KUKA KRL program: EPS_2_26115_SA7011_A_20260219035552.src

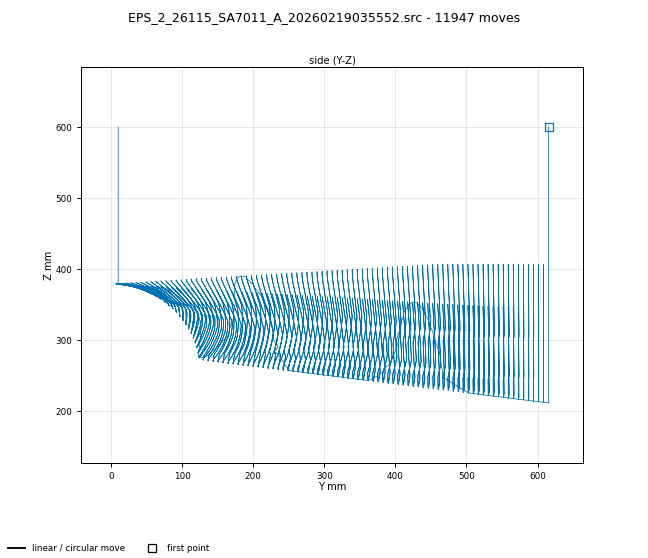
[picture p0: tool path of EPS_2_26115_SA7011_A_20260219035552.src, 11947 of 11949 moves have a stored position in this frame; points joined in program order, loops and branches not executed]
&ACCESS RVP
&REL 4
&COMMENT QRS 19112012
&PARAM EDITMASK = *
DEF PART()
EXT BAS (BAS_COMMAND :IN,REAL :IN )
INT I
BAS (#INITMOV,0 )

;KUKA QRS Post kuka4.cps  Date:22-06-2017 !

File_ID=3067

QRS_PRE_INIT()

;Init var - Until changes are made in qrs_pre_init
Outlet_Square_prg=0
Inlet_1_Square_prg=0
Inlet_2_Square_prg=0
Inlet_3_Square_prg=0
Inlet_4_Square_prg=0
Inlet_5_Square_prg=0

Outlet_1={X 0.000, Y 460.000, Z 306.500, B 0.000, E1 0.000 }
Inlet_1={X 0.000, Y 536.220, Z 246.500, B 0.000, E1 180.000 }
Outlet_1_type=201
Inlet_1_type=201
;QRS#1=Sidecore dimensions
;QRS#2=200-8" PVC SDR 35 Cut Back
;QRS#3=200-8" PVC SDR 35
;QRS#4=
;QRS#5=
;QRS#6=
;QRS#7=
;QRS#8=
;QRS#9=12-08 PSX
;QRS#10=12-08 PSX
;QRS#11=
;QRS#12=
;QRS#13=
;QRS#14=
;QRS#15=
;QRS#16=1220x127x686 2,25'
;QRS#17=EPS Height
;QRS#18=407
;QRS#19=*
;QRS#20= UPDATED VERSION 22-06-2017
;QRS#21=*
Outlet_Square=0100
Inlet_1_Square=0100
Inlet_2_Square=0
Inlet_3_Square=0
Inlet_4_Square=0
Inlet_5_Square=0
Mill_Square=1
Outlet_Square_Prg=214
Inlet_1_Square_prg=204

QRS_INIT()

$ADVANCE=5

; T1
PTP {E1 173.618,E2 173.618}
PTP {X 0,Y 615.492,A -85,B 0,C 180,E1 173.618,E2 173.618,E3 0,E4 0,E5 0,E6 0}
QRS_SPEED_INIT()
LIN {X 0,Y 615.492,Z 600,A -85,B 0,C 180,E1 173.618,E2 173.618,E3 0,E4 0,E5 0,E6 0} C_VEL
LIN {X 0,Y 615.492,Z 221.872,A -85,B 0,C 180,E1 173.618,E2 173.618} C_VEL
LIN {X 0,Y 615.492,Z 213.7,A -85,B 0,C 180,E1 173.618,E2 173.618} C_VEL
LIN {X 0,Y 615.48,Z 211.7,A -85,B 0,C 180,E1 173.432,E2 173.432} C_VEL
LIN {X 0,Y 615.497,Z 211.685,A -85,B 0,C 180,E1 170.801,E2 170.801} C_VEL
LIN {X 0,Y 615.486,Z 211.703,A -85,B 0,C 180,E1 168.139,E2 168.139} C_VEL
LIN {X 0,Y 615.448,Z 211.697,A -85,B 0,C 180,E1 165.45,E2 165.45} C_VEL
LIN {X 0,Y 615.468,Z 211.698,A -85,B 0,C 180,E1 162.729,E2 162.729} C_VEL
LIN {X 0,Y 615.465,Z 211.698,A -85,B 0,C 180,E1 159.966,E2 159.966} C_VEL
LIN {X 0,Y 615.489,Z 211.687,A -85,B 0,C 180,E1 157.155,E2 157.155} C_VEL
LIN {X 0,Y 615.481,Z 211.698,A -85,B 0,C 180,E1 154.284,E2 154.284} C_VEL
LIN {X 0,Y 615.466,Z 211.695,A -85,B 0,C 180,E1 151.554,E2 151.554} C_VEL
LIN {X 0,Y 615.449,Z 211.7,A -85,B 0,C 180,E1 148.921,E2 148.921} C_VEL
LIN {X 0,Y 615.453,Z 211.697,A -85,B 0,C 180,E1 146.471,E2 146.471} C_VEL
LIN {X 0,Y 615.489,Z 211.701,A -85,B 0,C 180,E1 144.167,E2 144.167} C_VEL
LIN {X 0,Y 615.48,Z 211.691,A -85,B 0,C 180,E1 141.931,E2 141.931} C_VEL
LIN {X 0,Y 615.493,Z 211.693,A -85,B 0,C 180,E1 139.394,E2 139.394} C_VEL
LIN {X 0,Y 615.44,Z 211.699,A -85,B 0,C 180,E1 136.751,E2 136.751} C_VEL
LIN {X 0,Y 615.483,Z 211.703,A -85,B 0,C 180,E1 133.997,E2 133.997} C_VEL
LIN {X 0,Y 615.468,Z 211.692,A -85,B 0,C 180,E1 131.476,E2 131.476} C_VEL
LIN {X 0,Y 615.489,Z 211.7,A -85,B 0,C 180,E1 128.905,E2 128.905} C_VEL
LIN {X 0,Y 615.472,Z 211.691,A -85,B 0,C 180,E1 126.426,E2 126.426} C_VEL
LIN {X 0,Y 615.493,Z 211.695,A -85,B 0,C 180,E1 125.616,E2 125.616} C_VEL
LIN {X 0,Y 615.455,Z 214.428,A -85,B 0,C 180,E1 123.239,E2 123.239} C_VEL
LIN {X 0,Y 615.428,Z 217.166,A -85,B 0,C 180,E1 120.923,E2 120.923} C_VEL
LIN {X 0,Y 615.496,Z 220.105,A -85,B 0,C 180,E1 118.451,E2 118.451} C_VEL
LIN {X 0,Y 615.445,Z 223.659,A -85,B 0,C 180,E1 115.718,E2 115.718} C_VEL
LIN {X 0,Y 615.442,Z 226.525,A -85,B 0,C 180,E1 113.558,E2 113.558} C_VEL
LIN {X 0,Y 615.45,Z 229.39,A -85,B 0,C 180,E1 111.434,E2 111.434} C_VEL
LIN {X 0,Y 615.496,Z 233.246,A -85,B 0,C 180,E1 108.606,E2 108.606} C_VEL
LIN {X 0,Y 615.457,Z 237.016,A -85,B 0,C 180,E1 105.906,E2 105.906} C_VEL
LIN {X 0,Y 615.495,Z 240.824,A -85,B 0,C 180,E1 103.201,E2 103.201} C_VEL
LIN {X 0,Y 615.481,Z 243.186,A -85,B 0,C 180,E1 101.548,E2 101.548} C_VEL
LIN {X 0,Y 615.491,Z 258.248,A -85,B 0,C 180,E1 101.193,E2 101.193} C_VEL
LIN {X 0,Y 615.496,Z 270.869,A -85,B 0,C 180,E1 100.753,E2 100.753} C_VEL
LIN {X 0,Y 615.468,Z 282.757,A -85,B 0,C 180,E1 100.195,E2 100.195} C_VEL
LIN {X 0,Y 615.497,Z 293.845,A -85,B 0,C 180,E1 99.53,E2 99.53} C_VEL
LIN {X 0,Y 615.498,Z 302.821,A -85,B 0,C 180,E1 98.868,E2 98.868} C_VEL
LIN {X 0,Y 615.498,Z 312.032,A -85,B 0,C 180,E1 98.041,E2 98.041} C_VEL
LIN {X 0,Y 615.499,Z 320.891,A -85,B 0,C 180,E1 97.058,E2 97.058} C_VEL
LIN {X 0,Y 615.497,Z 328.122,A -85,B 0,C 180,E1 96.063,E2 96.063} C_VEL
LIN {X 0,Y 615.497,Z 332.957,A -85,B 0,C 180,E1 95.241,E2 95.241} C_VEL
LIN {X 0,Y 615.493,Z 337.657,A -85,B 0,C 180,E1 94.257,E2 94.257} C_VEL
LIN {X 0,Y 615.495,Z 341.254,A -85,B 0,C 180,E1 93.273,E2 93.273} C_VEL
LIN {X 0,Y 615.496,Z 343.114,A -85,B 0,C 180,E1 92.618,E2 92.618} C_VEL
LIN {X 0,Y 615.497,Z 344.533,A -85,B 0,C 180,E1 91.963,E2 91.963} C_VEL
LIN {X 0,Y 615.496,Z 346.141,A -85,B 0,C 180,E1 90.654,E2 90.654} C_VEL
LIN {X 0,Y 615.494,Z 346.384,A -85,B 0,C 180,E1 90,E2 90} C_VEL
LIN {X 0,Y 615.495,Z 346.206,A -85,B 0,C 180,E1 89.346,E2 89.346} C_VEL
LIN {X 0,Y 615.496,Z 344.683,A -85,B 0,C 180,E1 88.037,E2 88.037} C_VEL
LIN {X 0,Y 615.498,Z 343.341,A -85,B 0,C 180,E1 87.382,E2 87.382} C_VEL
LIN {X 0,Y 615.496,Z 340.494,A -85,B 0,C 180,E1 86.399,E2 86.399} C_VEL
LIN {X 0,Y 615.498,Z 336.634,A -85,B 0,C 180,E1 85.416,E2 85.416} C_VEL
LIN {X 0,Y 615.498,Z 331.652,A -85,B 0,C 180,E1 84.43,E2 84.43} C_VEL
LIN {X 0,Y 615.497,Z 325.205,A -85,B 0,C 180,E1 83.417,E2 83.417} C_VEL
LIN {X 0,Y 615.497,Z 317.537,A -85,B 0,C 180,E1 82.455,E2 82.455} C_VEL
LIN {X 0,Y 615.498,Z 307.759,A -85,B 0,C 180,E1 81.464,E2 81.464} C_VEL
LIN {X 0,Y 615.498,Z 297.493,A -85,B 0,C 180,E1 80.636,E2 80.636} C_VEL
LIN {X 0,Y 615.469,Z 285.934,A -85,B 0,C 180,E1 79.888,E2 79.888} C_VEL
LIN {X 0,Y 615.492,Z 274.071,A -85,B 0,C 180,E1 79.293,E2 79.293} C_VEL
LIN {X 0,Y 615.486,Z 261.16,A -85,B 0,C 180,E1 78.807,E2 78.807} C_VEL
LIN {X 0,Y 615.486,Z 248.56,A -85,B 0,C 180,E1 78.473,E2 78.473} C_VEL
LIN {X 0,Y 615.483,Z 243.195,A -85,B 0,C 180,E1 78.369,E2 78.369} C_VEL
LIN {X 0,Y 615.466,Z 239.938,A -85,B 0,C 180,E1 76.077,E2 76.077} C_VEL
LIN {X 0,Y 615.49,Z 236.178,A -85,B 0,C 180,E1 73.413,E2 73.413} C_VEL
LIN {X 0,Y 615.472,Z 232.379,A -85,B 0,C 180,E1 70.662,E2 70.662} C_VEL
LIN {X 0,Y 615.458,Z 229.513,A -85,B 0,C 180,E1 68.567,E2 68.567} C_VEL
LIN {X 0,Y 615.465,Z 226.043,A -85,B 0,C 180,E1 65.997,E2 65.997} C_VEL
LIN {X 0,Y 615.494,Z 222.817,A -85,B 0,C 180,E1 63.556,E2 63.556} C_VEL
LIN {X 0,Y 615.475,Z 219.962,A -85,B 0,C 180,E1 61.341,E2 61.341} C_VEL
LIN {X 0,Y 615.429,Z 217.088,A -85,B 0,C 180,E1 58.924,E2 58.924} C_VEL
LIN {X 0,Y 615.471,Z 214.188,A -85,B 0,C 180,E1 56.469,E2 56.469} C_VEL
LIN {X 0,Y 615.496,Z 211.713,A -85,B 0,C 180,E1 54.385,E2 54.385} C_VEL
LIN {X 0,Y 615.485,Z 211.688,A -85,B 0,C 180,E1 51.931,E2 51.931} C_VEL
LIN {X 0,Y 615.487,Z 211.702,A -85,B 0,C 180,E1 49.393,E2 49.393} C_VEL
LIN {X 0,Y 615.455,Z 211.695,A -85,B 0,C 180,E1 46.752,E2 46.752} C_VEL
LIN {X 0,Y 615.466,Z 211.7,A -85,B 0,C 180,E1 43.995,E2 43.995} C_VEL
LIN {X 0,Y 615.447,Z 211.697,A -85,B 0,C 180,E1 41.477,E2 41.477} C_VEL
LIN {X 0,Y 615.49,Z 211.695,A -85,B 0,C 180,E1 38.904,E2 38.904} C_VEL
LIN {X 0,Y 615.486,Z 211.688,A -85,B 0,C 180,E1 36.425,E2 36.425} C_VEL
LIN {X 0,Y 615.492,Z 211.701,A -85,B 0,C 180,E1 34.022,E2 34.022} C_VEL
LIN {X 0,Y 615.442,Z 211.699,A -85,B 0,C 180,E1 31.688,E2 31.688} C_VEL
LIN {X 0,Y 615.439,Z 211.701,A -85,B 0,C 180,E1 29.409,E2 29.409} C_VEL
LIN {X 0,Y 615.471,Z 211.692,A -85,B 0,C 180,E1 26.445,E2 26.445} C_VEL
LIN {X 0,Y 615.478,Z 211.697,A -85,B 0,C 180,E1 24.006,E2 24.006} C_VEL
LIN {X 0,Y 615.471,Z 211.693,A -85,B 0,C 180,E1 21.433,E2 21.433} C_VEL
LIN {X 0,Y 615.491,Z 211.702,A -85,B 0,C 180,E1 18.605,E2 18.605} C_VEL
LIN {X 0,Y 615.434,Z 211.7,A -85,B 0,C 180,E1 15.907,E2 15.907} C_VEL
LIN {X 0,Y 615.495,Z 211.692,A -85,B 0,C 180,E1 13.201,E2 13.201} C_VEL
LIN {X 0,Y 615.472,Z 211.694,A -85,B 0,C 180,E1 10.527,E2 10.527} C_VEL
LIN {X 0,Y 615.473,Z 211.693,A -85,B 0,C 180,E1 7.876,E2 7.876} C_VEL
LIN {X 0,Y 615.497,Z 211.692,A -85,B 0,C 180,E1 5.241,E2 5.241} C_VEL
LIN {X 0,Y 615.437,Z 211.7,A -85,B 0,C 180,E1 2.618,E2 2.618} C_VEL
LIN {X 0,Y 615.477,Z 211.7,A -85,B 0,C 180,E1 0,E2 0} C_VEL
LIN {X 0,Y 615.483,Z 211.689,A -85,B 0,C 180,E1 -2.618,E2 -2.618} C_VEL
LIN {X 0,Y 615.496,Z 211.699,A -85,B 0,C 180,E1 -5.241,E2 -5.241} C_VEL
LIN {X 0,Y 615.466,Z 211.692,A -85,B 0,C 180,E1 -7.876,E2 -7.876} C_VEL
LIN {X 0,Y 615.485,Z 211.7,A -85,B 0,C 180,E1 -10.527,E2 -10.527} C_VEL
LIN {X 0,Y 615.437,Z 211.7,A -85,B 0,C 180,E1 -13.202,E2 -13.202} C_VEL
LIN {X 0,Y 615.495,Z 211.691,A -85,B 0,C 180,E1 -15.905,E2 -15.905} C_VEL
LIN {X 0,Y 615.481,Z 211.695,A -85,B 0,C 180,E1 -18.646,E2 -18.646} C_VEL
LIN {X 0,Y 615.468,Z 211.692,A -85,B 0,C 180,E1 -21.433,E2 -21.433} C_VEL
LIN {X 0,Y 615.475,Z 211.7,A -85,B 0,C 180,E1 -24.273,E2 -24.273} C_VEL
LIN {X 0,Y 615.436,Z 211.7,A -85,B 0,C 180,E1 -26.447,E2 -26.447} C_VEL
LIN {X 0,Y 615.452,Z 211.697,A -85,B 0,C 180,E1 -28.66,E2 -28.66} C_VEL
LIN {X 0,Y 615.488,Z 211.698,A -85,B 0,C 180,E1 -31.085,E2 -31.085} C_VEL
LIN {X 0,Y 615.495,Z 211.686,A -85,B 0,C 180,E1 -33.535,E2 -33.535} C_VEL
LIN {X 0,Y 615.464,Z 211.698,A -85,B 0,C 180,E1 -36.427,E2 -36.427} C_VEL
LIN {X 0,Y 615.458,Z 211.698,A -85,B 0,C 180,E1 -39.058,E2 -39.058} C_VEL
LIN {X 0,Y 615.484,Z 211.695,A -85,B 0,C 180,E1 -41.474,E2 -41.474} C_VEL
LIN {X 0,Y 615.463,Z 211.697,A -85,B 0,C 180,E1 -44.152,E2 -44.152} C_VEL
LIN {X 0,Y 615.484,Z 211.689,A -85,B 0,C 180,E1 -46.953,E2 -46.953} C_VEL
LIN {X 0,Y 615.479,Z 211.699,A -85,B 0,C 180,E1 -49.912,E2 -49.912} C_VEL
LIN {X 0,Y 615.446,Z 211.699,A -85,B 0,C 180,E1 -51.993,E2 -51.993} C_VEL
LIN {X 0,Y 615.46,Z 211.817,A -85,B 0,C 180,E1 -54.533,E2 -54.533} C_VEL
LIN {X 0,Y 615.471,Z 220.578,A -85,B 0,C 180,E1 -57.153,E2 -57.153} C_VEL
LIN {X 0,Y 615.452,Z 228.511,A -85,B 0,C 180,E1 -59.459,E2 -59.459} C_VEL
LIN {X 0,Y 615.48,Z 237.755,A -85,B 0,C 180,E1 -62.084,E2 -62.084} C_VEL
LIN {X 0,Y 615.488,Z 247.266,A -85,B 0,C 180,E1 -64.72,E2 -64.72} C_VEL
LIN {X 0,Y 615.475,Z 256.236,A -85,B 0,C 180,E1 -67.155,E2 -67.155} C_VEL
LIN {X 0,Y 615.49,Z 264.799,A -85,B 0,C 180,E1 -69.443,E2 -69.443} C_VEL
LIN {X 0,Y 615.49,Z 276.014,A -85,B 0,C 180,E1 -72.387,E2 -72.387} C_VEL
LIN {X 0,Y 615.479,Z 286.542,A -85,B 0,C 180,E1 -75.112,E2 -75.112} C_VEL
LIN {X 0,Y 615.444,Z 295.766,A -85,B 0,C 180,E1 -77.469,E2 -77.469} C_VEL
LIN {X 0,Y 615.498,Z 299.208,A -85,B 0,C 180,E1 -78.348,E2 -78.348} C_VEL
LIN {X 0,Y 615.497,Z 313.822,A -85,B 0,C 180,E1 -78.64,E2 -78.64} C_VEL
LIN {X 0,Y 615.451,Z 326.997,A -85,B 0,C 180,E1 -79.052,E2 -79.052} C_VEL
LIN {X 0,Y 615.438,Z 338.775,A -85,B 0,C 180,E1 -79.555,E2 -79.555} C_VEL
LIN {X 0,Y 615.482,Z 349.389,A -85,B 0,C 180,E1 -80.138,E2 -80.138} C_VEL
LIN {X 0,Y 615.498,Z 360.232,A -85,B 0,C 180,E1 -80.884,E2 -80.884} C_VEL
LIN {X 0,Y 615.497,Z 370.812,A -85,B 0,C 180,E1 -81.794,E2 -81.794} C_VEL
LIN {X 0,Y 615.498,Z 378.606,A -85,B 0,C 180,E1 -82.62,E2 -82.62} C_VEL
LIN {X 0,Y 615.496,Z 386.203,A -85,B 0,C 180,E1 -83.608,E2 -83.608} C_VEL
LIN {X 0,Y 615.498,Z 393.205,A -85,B 0,C 180,E1 -84.759,E2 -84.759} C_VEL
LIN {X 0,Y 615.494,Z 397.852,A -85,B 0,C 180,E1 -85.744,E2 -85.744} C_VEL
LIN {X 0,Y 615.494,Z 401.399,A -85,B 0,C 180,E1 -86.727,E2 -86.727} C_VEL
LIN {X 0,Y 615.497,Z 403.233,A -85,B 0,C 180,E1 -87.382,E2 -87.382} C_VEL
LIN {X 0,Y 615.5,Z 404.608,A -85,B 0,C 180,E1 -88.037,E2 -88.037} C_VEL
LIN {X 0,Y 615.496,Z 406.174,A -85,B 0,C 180,E1 -89.346,E2 -89.346} C_VEL
LIN {X 0,Y 615.494,Z 406.389,A -85,B 0,C 180,E1 -90,E2 -90} C_VEL
LIN {X 0,Y 615.495,Z 405.58,A -85,B 0,C 180,E1 -91.309,E2 -91.309} C_VEL
LIN {X 0,Y 615.5,Z 404.607,A -85,B 0,C 180,E1 -91.963,E2 -91.963} C_VEL
LIN {X 0,Y 615.497,Z 403.233,A -85,B 0,C 180,E1 -92.618,E2 -92.618} C_VEL
LIN {X 0,Y 615.496,Z 400.349,A -85,B 0,C 180,E1 -93.601,E2 -93.601} C_VEL
LIN {X 0,Y 615.498,Z 396.441,A -85,B 0,C 180,E1 -94.585,E2 -94.585} C_VEL
LIN {X 0,Y 615.499,Z 391.404,A -85,B 0,C 180,E1 -95.57,E2 -95.57} C_VEL
LIN {X 0,Y 615.497,Z 384.869,A -85,B 0,C 180,E1 -96.583,E2 -96.583} C_VEL
LIN {X 0,Y 615.497,Z 377.132,A -85,B 0,C 180,E1 -97.546,E2 -97.546} C_VEL
LIN {X 0,Y 615.498,Z 369.043,A -85,B 0,C 180,E1 -98.371,E2 -98.371} C_VEL
LIN {X 0,Y 615.499,Z 359.165,A -85,B 0,C 180,E1 -99.199,E2 -99.199} C_VEL
LIN {X 0,Y 615.471,Z 347.981,A -85,B 0,C 180,E1 -99.946,E2 -99.946} C_VEL
LIN {X 0,Y 615.437,Z 337.027,A -85,B 0,C 180,E1 -100.528,E2 -100.528} C_VEL
LIN {X 0,Y 615.457,Z 324.792,A -85,B 0,C 180,E1 -101.03,E2 -101.03} C_VEL
LIN {X 0,Y 615.499,Z 312.055,A -85,B 0,C 180,E1 -101.402,E2 -101.402} C_VEL
LIN {X 0,Y 615.498,Z 299.207,A -85,B 0,C 180,E1 -101.652,E2 -101.652} C_VEL
LIN {X 0,Y 615.454,Z 289.087,A -85,B 0,C 180,E1 -104.237,E2 -104.237} C_VEL
LIN {X 0,Y 615.491,Z 278.639,A -85,B 0,C 180,E1 -106.928,E2 -106.928} C_VEL
LIN {X 0,Y 615.482,Z 268.103,A -85,B 0,C 180,E1 -109.685,E2 -109.685} C_VEL
LIN {X 0,Y 615.49,Z 258.087,A -85,B 0,C 180,E1 -112.346,E2 -112.346} C_VEL
LIN {X 0,Y 615.477,Z 248.321,A -85,B 0,C 180,E1 -114.992,E2 -114.992} C_VEL
LIN {X 0,Y 615.492,Z 239.073,A -85,B 0,C 180,E1 -117.546,E2 -117.546} C_VEL
LIN {X 0,Y 615.456,Z 229.832,A -85,B 0,C 180,E1 -120.162,E2 -120.162} C_VEL
LIN {X 0,Y 615.445,Z 221.901,A -85,B 0,C 180,E1 -122.46,E2 -122.46} C_VEL
LIN {X 0,Y 615.492,Z 212.642,A -85,B 0,C 180,E1 -125.215,E2 -125.215} C_VEL
LIN {X 0,Y 615.455,Z 211.7,A -85,B 0,C 180,E1 -125.518,E2 -125.518} C_VEL
LIN {X 0,Y 615.448,Z 211.699,A -85,B 0,C 180,E1 -128.072,E2 -128.072} C_VEL
LIN {X 0,Y 615.491,Z 211.693,A -85,B 0,C 180,E1 -130.607,E2 -130.607} C_VEL
LIN {X 0,Y 615.48,Z 211.692,A -85,B 0,C 180,E1 -133.246,E2 -133.246} C_VEL
LIN {X 0,Y 615.459,Z 211.695,A -85,B 0,C 180,E1 -136.006,E2 -136.006} C_VEL
LIN {X 0,Y 615.48,Z 211.695,A -85,B 0,C 180,E1 -138.525,E2 -138.525} C_VEL
LIN {X 0,Y 615.446,Z 211.699,A -85,B 0,C 180,E1 -141.092,E2 -141.092} C_VEL
LIN {X 0,Y 615.462,Z 211.698,A -85,B 0,C 180,E1 -143.573,E2 -143.573} C_VEL
LIN {X 0,Y 615.495,Z 211.686,A -85,B 0,C 180,E1 -146.466,E2 -146.466} C_VEL
LIN {X 0,Y 615.491,Z 211.702,A -85,B 0,C 180,E1 -149.08,E2 -149.08} C_VEL
LIN {X 0,Y 615.45,Z 211.696,A -85,B 0,C 180,E1 -151.557,E2 -151.557} C_VEL
LIN {X 0,Y 615.471,Z 211.7,A -85,B 0,C 180,E1 -154.436,E2 -154.436} C_VEL
LIN {X 0,Y 615.469,Z 211.694,A -85,B 0,C 180,E1 -156.443,E2 -156.443} C_VEL
LIN {X 0,Y 615.466,Z 211.692,A -85,B 0,C 180,E1 -158.567,E2 -158.567} C_VEL
LIN {X 0,Y 615.483,Z 211.695,A -85,B 0,C 180,E1 -161.354,E2 -161.354} C_VEL
LIN {X 0,Y 615.495,Z 211.69,A -85,B 0,C 180,E1 -164.095,E2 -164.095} C_VEL
LIN {X 0,Y 615.442,Z 211.699,A -85,B 0,C 180,E1 -166.798,E2 -166.798} C_VEL
LIN {X 0,Y 615.48,Z 211.7,A -85,B 0,C 180,E1 -169.473,E2 -169.473} C_VEL
LIN {X 0,Y 615.467,Z 211.692,A -85,B 0,C 180,E1 -172.124,E2 -172.124} C_VEL
LIN {X 0,Y 615.495,Z 211.701,A -85,B 0,C 180,E1 -174.759,E2 -174.759} C_VEL
LIN {X 0,Y 615.484,Z 211.688,A -85,B 0,C 180,E1 -177.382,E2 -177.382} C_VEL
LIN {X 0,Y 615.479,Z 211.701,A -85,B 0,C 180,E1 -180,E2 -180} C_VEL
LIN {X 0,Y 615.435,Z 211.7,A -85,B 0,C 180,E1 -182.618,E2 -182.618} C_VEL
LIN {X 0,Y 615.497,Z 211.693,A -85,B 0,C 180,E1 -185.241,E2 -185.241} C_VEL
LIN {X 0,Y 615.48,Z 211.7,A -85,B 0,C 180,E1 -186.568,E2 -186.568} C_VEL
LIN {X 0,Y 614.812,Z 211.838,A -85,B 0,C 180,E1 -187.113,E2 -187.113} C_VEL
LIN {X 0,Y 611.989,Z 212.252,A -85,B 0,C 180,E1 -187.999,E2 -187.999} C_VEL
LIN {X 0,Y 609.599,Z 212.559,A -85,B 0,C 180,E1 -188.712,E2 -188.712} C_VEL
LIN {X 0,Y 608.558,Z 212.678,A -85,B 0,C 180,E1 -189.262,E2 -189.262} C_VEL
LIN {X 0,Y 608.466,Z 212.689,A -85,B 0,C 180,E1 -189.448,E2 -189.448} C_VEL
LIN {X 0,Y 608.458,Z 212.695,A -85,B 0,C 180,E1 -192,E2 -192} C_VEL
LIN {X 0,Y 608.422,Z 212.695,A -85,B 0,C 180,E1 -194.722,E2 -194.722} C_VEL
LIN {X 0,Y 608.428,Z 212.694,A -85,B 0,C 180,E1 -197.477,E2 -197.477} C_VEL
LIN {X 0,Y 608.433,Z 212.692,A -85,B 0,C 180,E1 -199.571,E2 -199.571} C_VEL
LIN {X 0,Y 608.483,Z 212.69,A -85,B 0,C 180,E1 -202.405,E2 -202.405} C_VEL
LIN {X 0,Y 608.457,Z 212.694,A -85,B 0,C 180,E1 -205.301,E2 -205.301} C_VEL
LIN {X 0,Y 608.437,Z 212.696,A -85,B 0,C 180,E1 -207.519,E2 -207.519} C_VEL
LIN {X 0,Y 608.406,Z 212.696,A -85,B 0,C 180,E1 -209.961,E2 -209.961} C_VEL
LIN {X 0,Y 608.47,Z 212.693,A -85,B 0,C 180,E1 -212.523,E2 -212.523} C_VEL
LIN {X 0,Y 608.439,Z 212.693,A -85,B 0,C 180,E1 -215.278,E2 -215.278} C_VEL
LIN {X 0,Y 608.465,Z 212.693,A -85,B 0,C 180,E1 -217.747,E2 -217.747} C_VEL
LIN {X 0,Y 608.449,Z 212.691,A -85,B 0,C 180,E1 -220.328,E2 -220.328} C_VEL
LIN {X 0,Y 608.424,Z 212.697,A -85,B 0,C 180,E1 -222.963,E2 -222.963} C_VEL
LIN {X 0,Y 608.441,Z 212.695,A -85,B 0,C 180,E1 -225.738,E2 -225.738} C_VEL
LIN {X 0,Y 608.442,Z 212.691,A -85,B 0,C 180,E1 -228.66,E2 -228.66} C_VEL
LIN {X 0,Y 608.471,Z 212.692,A -85,B 0,C 180,E1 -231.412,E2 -231.412} C_VEL
LIN {X 0,Y 608.451,Z 212.691,A -85,B 0,C 180,E1 -233.954,E2 -233.954} C_VEL
LIN {X 0,Y 608.437,Z 212.896,A -85,B 0,C 180,E1 -234.722,E2 -234.722} C_VEL
LIN {X 0,Y 608.403,Z 215.721,A -85,B 0,C 180,E1 -237.117,E2 -237.117} C_VEL
LIN {X 0,Y 608.435,Z 219.132,A -85,B 0,C 180,E1 -240.034,E2 -240.034} C_VEL
LIN {X 0,Y 608.39,Z 222.504,A -85,B 0,C 180,E1 -242.81,E2 -242.81} C_VEL
LIN {X 0,Y 608.413,Z 225.921,A -85,B 0,C 180,E1 -245.427,E2 -245.427} C_VEL
LIN {X 0,Y 608.385,Z 229.764,A -85,B 0,C 180,E1 -248.305,E2 -248.305} C_VEL
LIN {X 0,Y 608.388,Z 232.646,A -85,B 0,C 180,E1 -250.427,E2 -250.427} C_VEL
LIN {X 0,Y 608.417,Z 236.489,A -85,B 0,C 180,E1 -253.215,E2 -253.215} C_VEL
LIN {X 0,Y 608.394,Z 240.407,A -85,B 0,C 180,E1 -256.013,E2 -256.013} C_VEL
LIN {X 0,Y 608.423,Z 243.666,A -85,B 0,C 180,E1 -258.316,E2 -258.316} C_VEL
LIN {X 0,Y 608.535,Z 259.493,A -85,B 0,C 180,E1 -258.71,E2 -258.71} C_VEL
LIN {X 0,Y 608.518,Z 271.788,A -85,B 0,C 180,E1 -259.155,E2 -259.155} C_VEL
LIN {X 0,Y 608.467,Z 284.498,A -85,B 0,C 180,E1 -259.771,E2 -259.771} C_VEL
LIN {X 0,Y 608.487,Z 295.302,A -85,B 0,C 180,E1 -260.443,E2 -260.443} C_VEL
LIN {X 0,Y 608.477,Z 305.075,A -85,B 0,C 180,E1 -261.197,E2 -261.197} C_VEL
LIN {X 0,Y 608.46,Z 313.974,A -85,B 0,C 180,E1 -262.033,E2 -262.033} C_VEL
LIN {X 0,Y 608.465,Z 322.662,A -85,B 0,C 180,E1 -263.034,E2 -263.034} C_VEL
LIN {X 0,Y 608.439,Z 329.592,A -85,B 0,C 180,E1 -264.033,E2 -264.033} C_VEL
LIN {X 0,Y 608.436,Z 335.146,A -85,B 0,C 180,E1 -265.03,E2 -265.03} C_VEL
LIN {X 0,Y 608.434,Z 339.508,A -85,B 0,C 180,E1 -266.026,E2 -266.026} C_VEL
LIN {X 0,Y 608.425,Z 341.812,A -85,B 0,C 180,E1 -266.689,E2 -266.689} C_VEL
LIN {X 0,Y 608.425,Z 343.69,A -85,B 0,C 180,E1 -267.352,E2 -267.352} C_VEL
LIN {X 0,Y 608.442,Z 345.126,A -85,B 0,C 180,E1 -268.014,E2 -268.014} C_VEL
LIN {X 0,Y 608.439,Z 346.752,A -85,B 0,C 180,E1 -269.338,E2 -269.338} C_VEL
LIN {X 0,Y 608.434,Z 346.995,A -85,B 0,C 180,E1 -270,E2 -270} C_VEL
LIN {X 0,Y 608.438,Z 346.815,A -85,B 0,C 180,E1 -270.662,E2 -270.662} C_VEL
LIN {X 0,Y 608.441,Z 345.276,A -85,B 0,C 180,E1 -271.986,E2 -271.986} C_VEL
LIN {X 0,Y 608.427,Z 343.919,A -85,B 0,C 180,E1 -272.648,E2 -272.648} C_VEL
LIN {X 0,Y 608.449,Z 341.042,A -85,B 0,C 180,E1 -273.642,E2 -273.642} C_VEL
LIN {X 0,Y 608.433,Z 337.143,A -85,B 0,C 180,E1 -274.638,E2 -274.638} C_VEL
LIN {X 0,Y 608.449,Z 332.112,A -85,B 0,C 180,E1 -275.634,E2 -275.634} C_VEL
LIN {X 0,Y 608.442,Z 325.795,A -85,B 0,C 180,E1 -276.633,E2 -276.633} C_VEL
LIN {X 0,Y 608.475,Z 317.879,A -85,B 0,C 180,E1 -277.633,E2 -277.633} C_VEL
LIN {X 0,Y 608.472,Z 308.036,A -85,B 0,C 180,E1 -278.636,E2 -278.636} C_VEL
LIN {X 0,Y 608.481,Z 297.714,A -85,B 0,C 180,E1 -279.473,E2 -279.473} C_VEL
LIN {X 0,Y 608.466,Z 286.1,A -85,B 0,C 180,E1 -280.229,E2 -280.229} C_VEL
LIN {X 0,Y 608.509,Z 274.203,A -85,B 0,C 180,E1 -280.831,E2 -280.831} C_VEL
LIN {X 0,Y 608.529,Z 261.262,A -85,B 0,C 180,E1 -281.323,E2 -281.323} C_VEL
LIN {X 0,Y 608.535,Z 248.645,A -85,B 0,C 180,E1 -281.66,E2 -281.66} C_VEL
LIN {X 0,Y 608.427,Z 243.674,A -85,B 0,C 180,E1 -281.768,E2 -281.768} C_VEL
LIN {X 0,Y 608.418,Z 240.46,A -85,B 0,C 180,E1 -284.039,E2 -284.039} C_VEL
LIN {X 0,Y 608.418,Z 236.615,A -85,B 0,C 180,E1 -286.785,E2 -286.785} C_VEL
LIN {X 0,Y 608.395,Z 232.77,A -85,B 0,C 180,E1 -289.573,E2 -289.573} C_VEL
LIN {X 0,Y 608.389,Z 229.885,A -85,B 0,C 180,E1 -291.695,E2 -291.695} C_VEL
LIN {X 0,Y 608.416,Z 226.04,A -85,B 0,C 180,E1 -294.573,E2 -294.573} C_VEL
LIN {X 0,Y 608.398,Z 222.194,A -85,B 0,C 180,E1 -297.521,E2 -297.521} C_VEL
LIN {X 0,Y 608.437,Z 219.24,A -85,B 0,C 180,E1 -299.966,E2 -299.966} C_VEL
LIN {X 0,Y 608.397,Z 215.825,A -85,B 0,C 180,E1 -302.883,E2 -302.883} C_VEL
LIN {X 0,Y 608.436,Z 213.001,A -85,B 0,C 180,E1 -305.278,E2 -305.278} C_VEL
LIN {X 0,Y 608.478,Z 212.694,A -85,B 0,C 180,E1 -307.159,E2 -307.159} C_VEL
LIN {X 0,Y 608.449,Z 212.692,A -85,B 0,C 180,E1 -309.442,E2 -309.442} C_VEL
LIN {X 0,Y 608.469,Z 212.696,A -85,B 0,C 180,E1 -312.335,E2 -312.335} C_VEL
LIN {X 0,Y 608.414,Z 212.695,A -85,B 0,C 180,E1 -314.8,E2 -314.8} C_VEL
LIN {X 0,Y 608.468,Z 212.693,A -85,B 0,C 180,E1 -317.665,E2 -317.665} C_VEL
LIN {X 0,Y 608.447,Z 212.696,A -85,B 0,C 180,E1 -320.706,E2 -320.706} C_VEL
LIN {X 0,Y 608.451,Z 212.692,A -85,B 0,C 180,E1 -323.085,E2 -323.085} C_VEL
LIN {X 0,Y 608.472,Z 212.689,A -85,B 0,C 180,E1 -325.531,E2 -325.531} C_VEL
LIN {X 0,Y 608.459,Z 212.694,A -85,B 0,C 180,E1 -327.905,E2 -327.905} C_VEL
LIN {X 0,Y 608.419,Z 212.694,A -85,B 0,C 180,E1 -330.218,E2 -330.218} C_VEL
LIN {X 0,Y 608.461,Z 212.697,A -85,B 0,C 180,E1 -332.797,E2 -332.797} C_VEL
LIN {X 0,Y 608.45,Z 212.69,A -85,B 0,C 180,E1 -335.429,E2 -335.429} C_VEL
LIN {X 0,Y 608.463,Z 212.692,A -85,B 0,C 180,E1 -338.308,E2 -338.308} C_VEL
LIN {X 0,Y 608.476,Z 212.694,A -85,B 0,C 180,E1 -341.284,E2 -341.284} C_VEL
LIN {X 0,Y 608.416,Z 212.695,A -85,B 0,C 180,E1 -343.905,E2 -343.905} C_VEL
LIN {X 0,Y 608.464,Z 212.695,A -85,B 0,C 180,E1 -346.643,E2 -346.643} C_VEL
LIN {X 0,Y 608.453,Z 212.691,A -85,B 0,C 180,E1 -349.35,E2 -349.35} C_VEL
LIN {X 0,Y 608.469,Z 212.69,A -85,B 0,C 180,E1 -352.033,E2 -352.033} C_VEL
LIN {X 0,Y 608.473,Z 212.691,A -85,B 0,C 180,E1 -354.698,E2 -354.698} C_VEL
LIN {X 0,Y 608.435,Z 212.693,A -85,B 0,C 180,E1 -357.352,E2 -357.352} C_VEL
LIN {X 0,Y 608.469,Z 212.693,A -85,B 0,C 180,E1 -360,E2 -360} C_VEL
LIN {X 0,Y 608.475,Z 212.687,A -85,B 0,C 180,E1 -362.648,E2 -362.648} C_VEL
LIN {X 0,Y 608.473,Z 212.696,A -85,B 0,C 180,E1 -365.302,E2 -365.302} C_VEL
LIN {X 0,Y 608.437,Z 212.692,A -85,B 0,C 180,E1 -367.967,E2 -367.967} C_VEL
LIN {X 0,Y 608.45,Z 212.695,A -85,B 0,C 180,E1 -370.65,E2 -370.65} C_VEL
LIN {X 0,Y 608.432,Z 212.694,A -85,B 0,C 180,E1 -373.357,E2 -373.357} C_VEL
LIN {X 0,Y 608.461,Z 212.69,A -85,B 0,C 180,E1 -376.094,E2 -376.094} C_VEL
LIN {X 0,Y 608.454,Z 212.697,A -85,B 0,C 180,E1 -378.87,E2 -378.87} C_VEL
LIN {X 0,Y 608.461,Z 212.689,A -85,B 0,C 180,E1 -381.692,E2 -381.692} C_VEL
LIN {X 0,Y 608.429,Z 212.695,A -85,B 0,C 180,E1 -384.572,E2 -384.572} C_VEL
LIN {X 0,Y 608.455,Z 212.693,A -85,B 0,C 180,E1 -387.202,E2 -387.202} C_VEL
LIN {X 0,Y 608.445,Z 212.691,A -85,B 0,C 180,E1 -389.967,E2 -389.967} C_VEL
LIN {X 0,Y 608.462,Z 212.695,A -85,B 0,C 180,E1 -392.522,E2 -392.522} C_VEL
LIN {X 0,Y 608.442,Z 212.692,A -85,B 0,C 180,E1 -395.278,E2 -395.278} C_VEL
LIN {X 0,Y 608.456,Z 212.698,A -85,B 0,C 180,E1 -397.747,E2 -397.747} C_VEL
LIN {X 0,Y 608.404,Z 212.696,A -85,B 0,C 180,E1 -400.323,E2 -400.323} C_VEL
LIN {X 0,Y 608.457,Z 212.697,A -85,B 0,C 180,E1 -402.96,E2 -402.96} C_VEL
LIN {X 0,Y 608.445,Z 212.692,A -85,B 0,C 180,E1 -405.737,E2 -405.737} C_VEL
LIN {X 0,Y 608.452,Z 212.691,A -85,B 0,C 180,E1 -408.659,E2 -408.659} C_VEL
LIN {X 0,Y 608.435,Z 212.701,A -85,B 0,C 180,E1 -411.409,E2 -411.409} C_VEL
LIN {X 0,Y 608.429,Z 212.694,A -85,B 0,C 180,E1 -413.957,E2 -413.957} C_VEL
LIN {X 0,Y 608.446,Z 212.814,A -85,B 0,C 180,E1 -414.367,E2 -414.367} C_VEL
LIN {X 0,Y 608.529,Z 220.592,A -85,B 0,C 180,E1 -416.73,E2 -416.73} C_VEL
LIN {X 0,Y 608.481,Z 229.86,A -85,B 0,C 180,E1 -419.456,E2 -419.456} C_VEL
LIN {X 0,Y 608.494,Z 239.127,A -85,B 0,C 180,E1 -422.11,E2 -422.11} C_VEL
LIN {X 0,Y 608.479,Z 248.394,A -85,B 0,C 180,E1 -424.7,E2 -424.7} C_VEL
LIN {X 0,Y 608.48,Z 258.986,A -85,B 0,C 180,E1 -427.595,E2 -427.595} C_VEL
LIN {X 0,Y 608.457,Z 269.577,A -85,B 0,C 180,E1 -430.43,E2 -430.43} C_VEL
LIN {X 0,Y 608.45,Z 280.168,A -85,B 0,C 180,E1 -433.216,E2 -433.216} C_VEL
LIN {X 0,Y 608.437,Z 290.892,A -85,B 0,C 180,E1 -435.996,E2 -435.996} C_VEL
LIN {X 0,Y 608.437,Z 299.572,A -85,B 0,C 180,E1 -438.222,E2 -438.222} C_VEL
LIN {X 0,Y 608.55,Z 313.095,A -85,B 0,C 180,E1 -438.488,E2 -438.488} C_VEL
LIN {X 0,Y 608.486,Z 325.53,A -85,B 0,C 180,E1 -438.865,E2 -438.865} C_VEL
LIN {X 0,Y 608.444,Z 337.172,A -85,B 0,C 180,E1 -439.35,E2 -439.35} C_VEL
LIN {X 0,Y 608.471,Z 349.579,A -85,B 0,C 180,E1 -440.023,E2 -440.023} C_VEL
LIN {X 0,Y 608.483,Z 360.474,A -85,B 0,C 180,E1 -440.778,E2 -440.778} C_VEL
LIN {X 0,Y 608.475,Z 371.112,A -85,B 0,C 180,E1 -441.699,E2 -441.699} C_VEL
LIN {X 0,Y 608.471,Z 378.961,A -85,B 0,C 180,E1 -442.534,E2 -442.534} C_VEL
LIN {X 0,Y 608.461,Z 386.287,A -85,B 0,C 180,E1 -443.485,E2 -443.485} C_VEL
LIN {X 0,Y 608.451,Z 391.866,A -85,B 0,C 180,E1 -444.366,E2 -444.366} C_VEL
LIN {X 0,Y 608.432,Z 396.95,A -85,B 0,C 180,E1 -445.362,E2 -445.362} C_VEL
LIN {X 0,Y 608.449,Z 400.896,A -85,B 0,C 180,E1 -446.358,E2 -446.358} C_VEL
LIN {X 0,Y 608.425,Z 403.809,A -85,B 0,C 180,E1 -447.352,E2 -447.352} C_VEL
LIN {X 0,Y 608.444,Z 405.201,A -85,B 0,C 180,E1 -448.014,E2 -448.014} C_VEL
LIN {X 0,Y 608.438,Z 406.783,A -85,B 0,C 180,E1 -449.338,E2 -449.338} C_VEL
LIN {X 0,Y 608.434,Z 407,A -85,B 0,C 180,E1 -450,E2 -450} C_VEL
LIN {X 0,Y 608.448,Z 406.184,A -85,B 0,C 180,E1 -451.324,E2 -451.324} C_VEL
LIN {X 0,Y 608.444,Z 405.201,A -85,B 0,C 180,E1 -451.986,E2 -451.986} C_VEL
LIN {X 0,Y 608.425,Z 403.809,A -85,B 0,C 180,E1 -452.648,E2 -452.648} C_VEL
LIN {X 0,Y 608.449,Z 400.896,A -85,B 0,C 180,E1 -453.643,E2 -453.643} C_VEL
LIN {X 0,Y 608.432,Z 396.949,A -85,B 0,C 180,E1 -454.638,E2 -454.638} C_VEL
LIN {X 0,Y 608.438,Z 390.876,A -85,B 0,C 180,E1 -455.801,E2 -455.801} C_VEL
LIN {X 0,Y 608.462,Z 384.234,A -85,B 0,C 180,E1 -456.799,E2 -456.799} C_VEL
LIN {X 0,Y 608.456,Z 375.988,A -85,B 0,C 180,E1 -457.8,E2 -457.8} C_VEL
LIN {X 0,Y 608.472,Z 367.534,A -85,B 0,C 180,E1 -458.636,E2 -458.636} C_VEL
LIN {X 0,Y 608.48,Z 357.088,A -85,B 0,C 180,E1 -459.474,E2 -459.474} C_VEL
LIN {X 0,Y 608.482,Z 346.752,A -85,B 0,C 180,E1 -460.145,E2 -460.145} C_VEL
LIN {X 0,Y 608.463,Z 335.871,A -85,B 0,C 180,E1 -460.712,E2 -460.712} C_VEL
LIN {X 0,Y 608.492,Z 324.095,A -85,B 0,C 180,E1 -461.186,E2 -461.186} C_VEL
LIN {X 0,Y 608.551,Z 311.259,A -85,B 0,C 180,E1 -461.555,E2 -461.555} C_VEL
LIN {X 0,Y 608.439,Z 299.53,A -85,B 0,C 180,E1 -461.789,E2 -461.789} C_VEL
LIN {X 0,Y 608.405,Z 289.435,A -85,B 0,C 180,E1 -464.381,E2 -464.381} C_VEL
LIN {X 0,Y 608.45,Z 280.167,A -85,B 0,C 180,E1 -466.784,E2 -466.784} C_VEL
LIN {X 0,Y 608.457,Z 269.576,A -85,B 0,C 180,E1 -469.571,E2 -469.571} C_VEL
LIN {X 0,Y 608.464,Z 258.723,A -85,B 0,C 180,E1 -472.477,E2 -472.477} C_VEL
LIN {X 0,Y 608.479,Z 248.394,A -85,B 0,C 180,E1 -475.3,E2 -475.3} C_VEL
LIN {X 0,Y 608.496,Z 239.126,A -85,B 0,C 180,E1 -477.89,E2 -477.89} C_VEL
LIN {X 0,Y 608.481,Z 229.859,A -85,B 0,C 180,E1 -480.545,E2 -480.545} C_VEL
LIN {X 0,Y 608.528,Z 220.591,A -85,B 0,C 180,E1 -483.27,E2 -483.27} C_VEL
LIN {X 0,Y 608.438,Z 212.695,A -85,B 0,C 180,E1 -485.685,E2 -485.685} C_VEL
LIN {X 0,Y 608.443,Z 212.695,A -85,B 0,C 180,E1 -488.237,E2 -488.237} C_VEL
LIN {X 0,Y 608.448,Z 212.691,A -85,B 0,C 180,E1 -491.178,E2 -491.178} C_VEL
LIN {X 0,Y 608.466,Z 212.694,A -85,B 0,C 180,E1 -493.87,E2 -493.87} C_VEL
LIN {X 0,Y 608.483,Z 212.688,A -85,B 0,C 180,E1 -496.69,E2 -496.69} C_VEL
LIN {X 0,Y 608.45,Z 212.699,A -85,B 0,C 180,E1 -498.823,E2 -498.823} C_VEL
LIN {X 0,Y 608.417,Z 212.696,A -85,B 0,C 180,E1 -501.766,E2 -501.766} C_VEL
LIN {X 0,Y 608.45,Z 212.699,A -85,B 0,C 180,E1 -503.955,E2 -503.955} C_VEL
LIN {X 0,Y 608.47,Z 212.688,A -85,B 0,C 180,E1 -506.33,E2 -506.33} C_VEL
LIN {X 0,Y 608.451,Z 212.693,A -85,B 0,C 180,E1 -508.733,E2 -508.733} C_VEL
LIN {X 0,Y 608.445,Z 212.692,A -85,B 0,C 180,E1 -511.386,E2 -511.386} C_VEL
LIN {X 0,Y 608.47,Z 212.695,A -85,B 0,C 180,E1 -514.281,E2 -514.281} C_VEL
LIN {X 0,Y 608.429,Z 212.693,A -85,B 0,C 180,E1 -516.875,E2 -516.875} C_VEL
LIN {X 0,Y 608.469,Z 212.696,A -85,B 0,C 180,E1 -519.322,E2 -519.322} C_VEL
LIN {X 0,Y 608.452,Z 212.69,A -85,B 0,C 180,E1 -521.828,E2 -521.828} C_VEL
LIN {X 0,Y 608.463,Z 212.695,A -85,B 0,C 180,E1 -524.594,E2 -524.594} C_VEL
LIN {X 0,Y 608.435,Z 212.694,A -85,B 0,C 180,E1 -526.643,E2 -526.643} C_VEL
LIN {X 0,Y 608.446,Z 212.695,A -85,B 0,C 180,E1 -529.35,E2 -529.35} C_VEL
LIN {X 0,Y 608.438,Z 212.692,A -85,B 0,C 180,E1 -532.033,E2 -532.033} C_VEL
LIN {X 0,Y 608.472,Z 212.695,A -85,B 0,C 180,E1 -534.698,E2 -534.698} C_VEL
LIN {X 0,Y 608.476,Z 212.687,A -85,B 0,C 180,E1 -537.352,E2 -537.352} C_VEL
LIN {X 0,Y 608.471,Z 212.694,A -85,B 0,C 180,E1 -540,E2 -540} C_VEL
LIN {X 0,Y 608.433,Z 212.693,A -85,B 0,C 180,E1 -542.648,E2 -542.648} C_VEL
LIN {X 0,Y 608.472,Z 212.691,A -85,B 0,C 180,E1 -545.302,E2 -545.302} C_VEL
LIN {X 0,Y 608.44,Z 212.694,A -85,B 0,C 180,E1 -547.968,E2 -547.968} C_VEL
LIN {X 0,Y 608.466,Z 212.689,A -85,B 0,C 180,E1 -549.448,E2 -549.448} C_VEL
LIN {X 0,Y 607.778,Z 212.78,A -85,B 0,C 180,E1 -550,E2 -550} C_VEL
LIN {X 0,Y 604.922,Z 213.136,A -85,B 0,C 180,E1 -550.897,E2 -550.897} C_VEL
LIN {X 0,Y 602.52,Z 213.434,A -85,B 0,C 180,E1 -551.619,E2 -551.619} C_VEL
LIN {X 0,Y 601.488,Z 213.561,A -85,B 0,C 180,E1 -552.175,E2 -552.175} C_VEL
LIN {X 0,Y 601.403,Z 213.57,A -85,B 0,C 180,E1 -552.364,E2 -552.364} C_VEL
LIN {X 0,Y 601.394,Z 213.572,A -85,B 0,C 180,E1 -554.898,E2 -554.898} C_VEL
LIN {X 0,Y 601.373,Z 213.572,A -85,B 0,C 180,E1 -557.689,E2 -557.689} C_VEL
LIN {X 0,Y 601.434,Z 213.57,A -85,B 0,C 180,E1 -560.522,E2 -560.522} C_VEL
LIN {X 0,Y 601.4,Z 213.571,A -85,B 0,C 180,E1 -563.411,E2 -563.411} C_VEL
LIN {X 0,Y 601.409,Z 213.571,A -85,B 0,C 180,E1 -565.865,E2 -565.865} C_VEL
LIN {X 0,Y 601.424,Z 213.569,A -85,B 0,C 180,E1 -568.627,E2 -568.627} C_VEL
LIN {X 0,Y 601.393,Z 213.57,A -85,B 0,C 180,E1 -571.728,E2 -571.728} C_VEL
LIN {X 0,Y 601.424,Z 213.573,A -85,B 0,C 180,E1 -574.119,E2 -574.119} C_VEL
LIN {X 0,Y 601.402,Z 213.569,A -85,B 0,C 180,E1 -576.583,E2 -576.583} C_VEL
LIN {X 0,Y 601.409,Z 213.575,A -85,B 0,C 180,E1 -579.127,E2 -579.127} C_VEL
LIN {X 0,Y 601.414,Z 213.567,A -85,B 0,C 180,E1 -581.766,E2 -581.766} C_VEL
LIN {X 0,Y 601.402,Z 213.573,A -85,B 0,C 180,E1 -584.532,E2 -584.532} C_VEL
LIN {X 0,Y 601.388,Z 213.573,A -85,B 0,C 180,E1 -587.412,E2 -587.412} C_VEL
LIN {X 0,Y 601.406,Z 213.569,A -85,B 0,C 180,E1 -590.004,E2 -590.004} C_VEL
LIN {X 0,Y 601.44,Z 213.568,A -85,B 0,C 180,E1 -592.618,E2 -592.618} C_VEL
LIN {X 0,Y 601.375,Z 213.806,A -85,B 0,C 180,E1 -594.891,E2 -594.891} C_VEL
LIN {X 0,Y 601.349,Z 216.8,A -85,B 0,C 180,E1 -597.479,E2 -597.479} C_VEL
LIN {X 0,Y 601.349,Z 219.549,A -85,B 0,C 180,E1 -599.865,E2 -599.865} C_VEL
LIN {X 0,Y 601.314,Z 222.827,A -85,B 0,C 180,E1 -602.657,E2 -602.657} C_VEL
LIN {X 0,Y 601.327,Z 225.921,A -85,B 0,C 180,E1 -605.118,E2 -605.118} C_VEL
LIN {X 0,Y 601.32,Z 229.764,A -85,B 0,C 180,E1 -608.037,E2 -608.037} C_VEL
LIN {X 0,Y 601.297,Z 232.647,A -85,B 0,C 180,E1 -610.187,E2 -610.187} C_VEL
LIN {X 0,Y 601.295,Z 235.529,A -85,B 0,C 180,E1 -612.308,E2 -612.308} C_VEL
LIN {X 0,Y 601.31,Z 238.412,A -85,B 0,C 180,E1 -614.406,E2 -614.406} C_VEL
LIN {X 0,Y 601.321,Z 242.256,A -85,B 0,C 180,E1 -617.169,E2 -617.169} C_VEL
LIN {X 0,Y 601.328,Z 243.667,A -85,B 0,C 180,E1 -618.176,E2 -618.176} C_VEL
LIN {X 0,Y 601.598,Z 247.38,A -85,B 0,C 180,E1 -618.267,E2 -618.267} C_VEL
LIN {X 0,Y 601.565,Z 259.674,A -85,B 0,C 180,E1 -618.583,E2 -618.583} C_VEL
LIN {X 0,Y 601.547,Z 272.824,A -85,B 0,C 180,E1 -619.072,E2 -619.072} C_VEL
LIN {X 0,Y 601.477,Z 284.51,A -85,B 0,C 180,E1 -619.65,E2 -619.65} C_VEL
LIN {X 0,Y 601.458,Z 295.308,A -85,B 0,C 180,E1 -620.33,E2 -620.33} C_VEL
LIN {X 0,Y 601.435,Z 305.082,A -85,B 0,C 180,E1 -621.093,E2 -621.093} C_VEL
LIN {X 0,Y 601.407,Z 313.979,A -85,B 0,C 180,E1 -621.939,E2 -621.939} C_VEL
LIN {X 0,Y 601.407,Z 322.666,A -85,B 0,C 180,E1 -622.952,E2 -622.952} C_VEL
LIN {X 0,Y 601.361,Z 329.596,A -85,B 0,C 180,E1 -623.962,E2 -623.962} C_VEL
LIN {X 0,Y 601.345,Z 335.148,A -85,B 0,C 180,E1 -624.971,E2 -624.971} C_VEL
LIN {X 0,Y 601.346,Z 339.51,A -85,B 0,C 180,E1 -625.979,E2 -625.979} C_VEL
LIN {X 0,Y 601.344,Z 341.814,A -85,B 0,C 180,E1 -626.65,E2 -626.65} C_VEL
LIN {X 0,Y 601.324,Z 343.692,A -85,B 0,C 180,E1 -627.32,E2 -627.32} C_VEL
LIN {X 0,Y 601.341,Z 345.127,A -85,B 0,C 180,E1 -627.991,E2 -627.991} C_VEL
LIN {X 0,Y 601.339,Z 346.752,A -85,B 0,C 180,E1 -629.33,E2 -629.33} C_VEL
LIN {X 0,Y 601.335,Z 346.996,A -85,B 0,C 180,E1 -630,E2 -630} C_VEL
LIN {X 0,Y 601.339,Z 346.815,A -85,B 0,C 180,E1 -630.67,E2 -630.67} C_VEL
LIN {X 0,Y 601.34,Z 345.276,A -85,B 0,C 180,E1 -632.009,E2 -632.009} C_VEL
LIN {X 0,Y 601.326,Z 343.917,A -85,B 0,C 180,E1 -632.679,E2 -632.679} C_VEL
LIN {X 0,Y 601.368,Z 341.04,A -85,B 0,C 180,E1 -633.685,E2 -633.685} C_VEL
LIN {X 0,Y 601.337,Z 337.141,A -85,B 0,C 180,E1 -634.693,E2 -634.693} C_VEL
LIN {X 0,Y 601.373,Z 332.11,A -85,B 0,C 180,E1 -635.701,E2 -635.701} C_VEL
LIN {X 0,Y 601.382,Z 325.792,A -85,B 0,C 180,E1 -636.711,E2 -636.711} C_VEL
LIN {X 0,Y 601.396,Z 317.874,A -85,B 0,C 180,E1 -637.723,E2 -637.723} C_VEL
LIN {X 0,Y 601.437,Z 308.03,A -85,B 0,C 180,E1 -638.738,E2 -638.738} C_VEL
LIN {X 0,Y 601.448,Z 297.709,A -85,B 0,C 180,E1 -639.585,E2 -639.585} C_VEL
LIN {X 0,Y 601.479,Z 286.089,A -85,B 0,C 180,E1 -640.349,E2 -640.349} C_VEL
LIN {X 0,Y 601.524,Z 274.192,A -85,B 0,C 180,E1 -640.959,E2 -640.959} C_VEL
LIN {X 0,Y 601.551,Z 261.247,A -85,B 0,C 180,E1 -641.456,E2 -641.456} C_VEL
LIN {X 0,Y 601.604,Z 248.622,A -85,B 0,C 180,E1 -641.797,E2 -641.797} C_VEL
LIN {X 0,Y 601.331,Z 243.673,A -85,B 0,C 180,E1 -641.909,E2 -641.909} C_VEL
LIN {X 0,Y 601.317,Z 240.459,A -85,B 0,C 180,E1 -644.208,E2 -644.208} C_VEL
LIN {X 0,Y 601.334,Z 236.614,A -85,B 0,C 180,E1 -646.989,E2 -646.989} C_VEL
LIN {X 0,Y 601.301,Z 232.769,A -85,B 0,C 180,E1 -649.813,E2 -649.813} C_VEL
LIN {X 0,Y 601.322,Z 229.885,A -85,B 0,C 180,E1 -651.963,E2 -651.963} C_VEL
LIN {X 0,Y 601.331,Z 226.039,A -85,B 0,C 180,E1 -654.882,E2 -654.882} C_VEL
LIN {X 0,Y 601.32,Z 222.899,A -85,B 0,C 180,E1 -657.344,E2 -657.344} C_VEL
LIN {X 0,Y 601.352,Z 219.647,A -85,B 0,C 180,E1 -660.168,E2 -660.168} C_VEL
LIN {X 0,Y 601.335,Z 216.694,A -85,B 0,C 180,E1 -662.702,E2 -662.702} C_VEL
LIN {X 0,Y 601.371,Z 213.909,A -85,B 0,C 180,E1 -665.108,E2 -665.108} C_VEL
LIN {X 0,Y 601.399,Z 213.57,A -85,B 0,C 180,E1 -666.583,E2 -666.583} C_VEL
LIN {X 0,Y 601.418,Z 213.571,A -85,B 0,C 180,E1 -669.126,E2 -669.126} C_VEL
LIN {X 0,Y 601.425,Z 213.566,A -85,B 0,C 180,E1 -671.765,E2 -671.765} C_VEL
LIN {X 0,Y 601.4,Z 213.57,A -85,B 0,C 180,E1 -674.532,E2 -674.532} C_VEL
LIN {X 0,Y 601.41,Z 213.575,A -85,B 0,C 180,E1 -677.41,E2 -677.41} C_VEL
LIN {X 0,Y 601.403,Z 213.568,A -85,B 0,C 180,E1 -680.004,E2 -680.004} C_VEL
LIN {X 0,Y 601.438,Z 213.572,A -85,B 0,C 180,E1 -682.618,E2 -682.618} C_VEL
LIN {X 0,Y 601.407,Z 213.568,A -85,B 0,C 180,E1 -685.067,E2 -685.067} C_VEL
LIN {X 0,Y 601.436,Z 213.569,A -85,B 0,C 180,E1 -687.484,E2 -687.484} C_VEL
LIN {X 0,Y 601.373,Z 213.574,A -85,B 0,C 180,E1 -689.861,E2 -689.861} C_VEL
LIN {X 0,Y 601.372,Z 213.572,A -85,B 0,C 180,E1 -692.13,E2 -692.13} C_VEL
LIN {X 0,Y 601.431,Z 213.57,A -85,B 0,C 180,E1 -694.382,E2 -694.382} C_VEL
LIN {X 0,Y 601.421,Z 213.569,A -85,B 0,C 180,E1 -696.59,E2 -696.59} C_VEL
LIN {X 0,Y 601.434,Z 213.57,A -85,B 0,C 180,E1 -699.478,E2 -699.478} C_VEL
LIN {X 0,Y 601.374,Z 213.572,A -85,B 0,C 180,E1 -702.311,E2 -702.311} C_VEL
LIN {X 0,Y 601.393,Z 213.573,A -85,B 0,C 180,E1 -705.102,E2 -705.102} C_VEL
LIN {X 0,Y 601.411,Z 213.57,A -85,B 0,C 180,E1 -707.857,E2 -707.857} C_VEL
LIN {X 0,Y 601.424,Z 213.566,A -85,B 0,C 180,E1 -710.584,E2 -710.584} C_VEL
LIN {X 0,Y 601.435,Z 213.572,A -85,B 0,C 180,E1 -713.345,E2 -713.345} C_VEL
LIN {X 0,Y 601.371,Z 213.572,A -85,B 0,C 180,E1 -715.979,E2 -715.979} C_VEL
LIN {X 0,Y 601.417,Z 213.572,A -85,B 0,C 180,E1 -718.661,E2 -718.661} C_VEL
LIN {X 0,Y 601.398,Z 213.57,A -85,B 0,C 180,E1 -721.339,E2 -721.339} C_VEL
LIN {X 0,Y 601.422,Z 213.57,A -85,B 0,C 180,E1 -723.35,E2 -723.35} C_VEL
LIN {X 0,Y 601.406,Z 213.568,A -85,B 0,C 180,E1 -726.037,E2 -726.037} C_VEL
LIN {X 0,Y 601.415,Z 213.575,A -85,B 0,C 180,E1 -728.738,E2 -728.738} C_VEL
LIN {X 0,Y 601.396,Z 213.569,A -85,B 0,C 180,E1 -731.459,E2 -731.459} C_VEL
LIN {X 0,Y 601.417,Z 213.569,A -85,B 0,C 180,E1 -734.206,E2 -734.206} C_VEL
LIN {X 0,Y 601.415,Z 213.571,A -85,B 0,C 180,E1 -736.986,E2 -736.986} C_VEL
LIN {X 0,Y 601.406,Z 213.568,A -85,B 0,C 180,E1 -739.809,E2 -739.809} C_VEL
LIN {X 0,Y 601.413,Z 213.571,A -85,B 0,C 180,E1 -742.683,E2 -742.683} C_VEL
LIN {X 0,Y 601.378,Z 213.571,A -85,B 0,C 180,E1 -744.88,E2 -744.88} C_VEL
LIN {X 0,Y 601.398,Z 213.574,A -85,B 0,C 180,E1 -747.359,E2 -747.359} C_VEL
LIN {X 0,Y 601.405,Z 213.568,A -85,B 0,C 180,E1 -750.165,E2 -750.165} C_VEL
LIN {X 0,Y 601.423,Z 213.573,A -85,B 0,C 180,E1 -752.715,E2 -752.715} C_VEL
LIN {X 0,Y 601.392,Z 213.57,A -85,B 0,C 180,E1 -755.111,E2 -755.111} C_VEL
LIN {X 0,Y 601.432,Z 213.568,A -85,B 0,C 180,E1 -757.419,E2 -757.419} C_VEL
LIN {X 0,Y 601.376,Z 213.573,A -85,B 0,C 180,E1 -759.998,E2 -759.998} C_VEL
LIN {X 0,Y 601.387,Z 213.575,A -85,B 0,C 180,E1 -762.673,E2 -762.673} C_VEL
LIN {X 0,Y 601.401,Z 213.569,A -85,B 0,C 180,E1 -765.479,E2 -765.479} C_VEL
LIN {X 0,Y 601.422,Z 213.569,A -85,B 0,C 180,E1 -768.407,E2 -768.407} C_VEL
LIN {X 0,Y 601.402,Z 213.57,A -85,B 0,C 180,E1 -770.872,E2 -770.872} C_VEL
LIN {X 0,Y 601.396,Z 213.576,A -85,B 0,C 180,E1 -773.416,E2 -773.416} C_VEL
LIN {X 0,Y 601.403,Z 213.688,A -85,B 0,C 180,E1 -774.158,E2 -774.158} C_VEL
LIN {X 0,Y 601.544,Z 219.268,A -85,B 0,C 180,E1 -775.889,E2 -775.889} C_VEL
LIN {X 0,Y 601.566,Z 228.022,A -85,B 0,C 180,E1 -778.523,E2 -778.523} C_VEL
LIN {X 0,Y 601.479,Z 237.803,A -85,B 0,C 180,E1 -781.375,E2 -781.375} C_VEL
LIN {X 0,Y 601.478,Z 247.454,A -85,B 0,C 180,E1 -784.12,E2 -784.12} C_VEL
LIN {X 0,Y 601.466,Z 256.338,A -85,B 0,C 180,E1 -786.592,E2 -786.592} C_VEL
LIN {X 0,Y 601.431,Z 266.929,A -85,B 0,C 180,E1 -789.478,E2 -789.478} C_VEL
LIN {X 0,Y 601.4,Z 277.52,A -85,B 0,C 180,E1 -792.312,E2 -792.312} C_VEL
LIN {X 0,Y 601.366,Z 288.112,A -85,B 0,C 180,E1 -795.101,E2 -795.101} C_VEL
LIN {X 0,Y 601.342,Z 298.703,A -85,B 0,C 180,E1 -797.856,E2 -797.856} C_VEL
LIN {X 0,Y 601.372,Z 299.53,A -85,B 0,C 180,E1 -798.071,E2 -798.071} C_VEL
LIN {X 0,Y 601.618,Z 311.268,A -85,B 0,C 180,E1 -798.311,E2 -798.311} C_VEL
LIN {X 0,Y 601.533,Z 324.353,A -85,B 0,C 180,E1 -798.692,E2 -798.692} C_VEL
LIN {X 0,Y 601.48,Z 335.262,A -85,B 0,C 180,E1 -799.133,E2 -799.133} C_VEL
LIN {X 0,Y 601.473,Z 346.756,A -85,B 0,C 180,E1 -799.736,E2 -799.736} C_VEL
LIN {X 0,Y 601.462,Z 358.253,A -85,B 0,C 180,E1 -800.5,E2 -800.5} C_VEL
LIN {X 0,Y 601.436,Z 367.537,A -85,B 0,C 180,E1 -801.262,E2 -801.262} C_VEL
LIN {X 0,Y 601.4,Z 375.99,A -85,B 0,C 180,E1 -802.108,E2 -802.108} C_VEL
LIN {X 0,Y 601.382,Z 384.236,A -85,B 0,C 180,E1 -803.12,E2 -803.12} C_VEL
LIN {X 0,Y 601.373,Z 390.877,A -85,B 0,C 180,E1 -804.131,E2 -804.131} C_VEL
LIN {X 0,Y 601.336,Z 396.95,A -85,B 0,C 180,E1 -805.307,E2 -805.307} C_VEL
LIN {X 0,Y 601.368,Z 400.896,A -85,B 0,C 180,E1 -806.315,E2 -806.315} C_VEL
LIN {X 0,Y 601.325,Z 403.809,A -85,B 0,C 180,E1 -807.321,E2 -807.321} C_VEL
LIN {X 0,Y 601.343,Z 405.202,A -85,B 0,C 180,E1 -807.991,E2 -807.991} C_VEL
LIN {X 0,Y 601.339,Z 406.784,A -85,B 0,C 180,E1 -809.33,E2 -809.33} C_VEL
LIN {X 0,Y 601.335,Z 407,A -85,B 0,C 180,E1 -810,E2 -810} C_VEL
LIN {X 0,Y 601.347,Z 406.184,A -85,B 0,C 180,E1 -811.339,E2 -811.339} C_VEL
LIN {X 0,Y 601.343,Z 405.201,A -85,B 0,C 180,E1 -812.009,E2 -812.009} C_VEL
LIN {X 0,Y 601.325,Z 403.809,A -85,B 0,C 180,E1 -812.68,E2 -812.68} C_VEL
LIN {X 0,Y 601.368,Z 400.896,A -85,B 0,C 180,E1 -813.685,E2 -813.685} C_VEL
LIN {X 0,Y 601.336,Z 396.949,A -85,B 0,C 180,E1 -814.693,E2 -814.693} C_VEL
LIN {X 0,Y 601.373,Z 390.876,A -85,B 0,C 180,E1 -815.869,E2 -815.869} C_VEL
LIN {X 0,Y 601.382,Z 384.234,A -85,B 0,C 180,E1 -816.88,E2 -816.88} C_VEL
LIN {X 0,Y 601.4,Z 375.988,A -85,B 0,C 180,E1 -817.892,E2 -817.892} C_VEL
LIN {X 0,Y 601.436,Z 367.534,A -85,B 0,C 180,E1 -818.738,E2 -818.738} C_VEL
LIN {X 0,Y 601.447,Z 357.089,A -85,B 0,C 180,E1 -819.585,E2 -819.585} C_VEL
LIN {X 0,Y 601.473,Z 346.753,A -85,B 0,C 180,E1 -820.265,E2 -820.265} C_VEL
LIN {X 0,Y 601.481,Z 335.248,A -85,B 0,C 180,E1 -820.868,E2 -820.868} C_VEL
LIN {X 0,Y 601.527,Z 322.334,A -85,B 0,C 180,E1 -821.375,E2 -821.375} C_VEL
LIN {X 0,Y 601.615,Z 309.43,A -85,B 0,C 180,E1 -821.732,E2 -821.732} C_VEL
LIN {X 0,Y 601.373,Z 299.53,A -85,B 0,C 180,E1 -821.93,E2 -821.93} C_VEL
LIN {X 0,Y 601.369,Z 289.435,A -85,B 0,C 180,E1 -824.552,E2 -824.552} C_VEL
LIN {X 0,Y 601.395,Z 278.843,A -85,B 0,C 180,E1 -827.338,E2 -827.338} C_VEL
LIN {X 0,Y 601.421,Z 268.252,A -85,B 0,C 180,E1 -830.165,E2 -830.165} C_VEL
LIN {X 0,Y 601.434,Z 258.985,A -85,B 0,C 180,E1 -832.682,E2 -832.682} C_VEL
LIN {X 0,Y 601.463,Z 249.717,A -85,B 0,C 180,E1 -835.246,E2 -835.246} C_VEL
LIN {X 0,Y 601.504,Z 240.45,A -85,B 0,C 180,E1 -837.864,E2 -837.864} C_VEL
LIN {X 0,Y 601.506,Z 231.183,A -85,B 0,C 180,E1 -840.548,E2 -840.548} C_VEL
LIN {X 0,Y 601.584,Z 221.915,A -85,B 0,C 180,E1 -843.304,E2 -843.304} C_VEL
LIN {X 0,Y 601.585,Z 215.919,A -85,B 0,C 180,E1 -845.137,E2 -845.137} C_VEL
LIN {X 0,Y 601.402,Z 213.573,A -85,B 0,C 180,E1 -845.932,E2 -845.932} C_VEL
LIN {X 0,Y 601.407,Z 213.575,A -85,B 0,C 180,E1 -848.468,E2 -848.468} C_VEL
LIN {X 0,Y 601.412,Z 213.568,A -85,B 0,C 180,E1 -850.875,E2 -850.875} C_VEL
LIN {X 0,Y 601.432,Z 213.571,A -85,B 0,C 180,E1 -853.586,E2 -853.586} C_VEL
LIN {X 0,Y 601.433,Z 213.565,A -85,B 0,C 180,E1 -856.428,E2 -856.428} C_VEL
LIN {X 0,Y 601.401,Z 213.572,A -85,B 0,C 180,E1 -859.124,E2 -859.124} C_VEL
LIN {X 0,Y 601.37,Z 213.574,A -85,B 0,C 180,E1 -861.728,E2 -861.728} C_VEL
LIN {X 0,Y 601.391,Z 213.574,A -85,B 0,C 180,E1 -864.245,E2 -864.245} C_VEL
LIN {X 0,Y 601.43,Z 213.565,A -85,B 0,C 180,E1 -866.687,E2 -866.687} C_VEL
LIN {X 0,Y 601.408,Z 213.575,A -85,B 0,C 180,E1 -869.057,E2 -869.057} C_VEL
LIN {X 0,Y 601.405,Z 213.569,A -85,B 0,C 180,E1 -871.372,E2 -871.372} C_VEL
LIN {X 0,Y 601.403,Z 213.575,A -85,B 0,C 180,E1 -874.136,E2 -874.136} C_VEL
LIN {X 0,Y 601.388,Z 213.571,A -85,B 0,C 180,E1 -876.588,E2 -876.588} C_VEL
LIN {X 0,Y 601.434,Z 213.571,A -85,B 0,C 180,E1 -879.478,E2 -879.478} C_VEL
LIN {X 0,Y 601.403,Z 213.57,A -85,B 0,C 180,E1 -882.312,E2 -882.312} C_VEL
LIN {X 0,Y 601.409,Z 213.575,A -85,B 0,C 180,E1 -884.409,E2 -884.409} C_VEL
LIN {X 0,Y 601.4,Z 213.572,A -85,B 0,C 180,E1 -886.484,E2 -886.484} C_VEL
LIN {X 0,Y 601.384,Z 213.573,A -85,B 0,C 180,E1 -889.223,E2 -889.223} C_VEL
LIN {X 0,Y 601.413,Z 213.568,A -85,B 0,C 180,E1 -891.939,E2 -891.939} C_VEL
LIN {X 0,Y 601.406,Z 213.568,A -85,B 0,C 180,E1 -893.963,E2 -893.963} C_VEL
LIN {X 0,Y 601.425,Z 213.571,A -85,B 0,C 180,E1 -896.65,E2 -896.65} C_VEL
LIN {X 0,Y 601.445,Z 213.564,A -85,B 0,C 180,E1 -899.331,E2 -899.331} C_VEL
LIN {X 0,Y 601.397,Z 213.571,A -85,B 0,C 180,E1 -902.009,E2 -902.009} C_VEL
LIN {X 0,Y 601.4,Z 213.572,A -85,B 0,C 180,E1 -904.692,E2 -904.692} C_VEL
LIN {X 0,Y 601.441,Z 213.564,A -85,B 0,C 180,E1 -907.385,E2 -907.385} C_VEL
LIN {X 0,Y 601.429,Z 213.573,A -85,B 0,C 180,E1 -910.095,E2 -910.095} C_VEL
LIN {X 0,Y 601.403,Z 213.57,A -85,B 0,C 180,E1 -912.364,E2 -912.364} C_VEL
LIN {X 0,Y 600.731,Z 213.653,A -85,B 0,C 180,E1 -912.923,E2 -912.923} C_VEL
LIN {X 0,Y 597.873,Z 214.012,A -85,B 0,C 180,E1 -913.83,E2 -913.83} C_VEL
LIN {X 0,Y 595.46,Z 214.314,A -85,B 0,C 180,E1 -914.56,E2 -914.56} C_VEL
LIN {X 0,Y 594.421,Z 214.444,A -85,B 0,C 180,E1 -915.123,E2 -915.123} C_VEL
LIN {X 0,Y 594.336,Z 214.451,A -85,B 0,C 180,E1 -915.314,E2 -915.314} C_VEL
LIN {X 0,Y 594.33,Z 214.449,A -85,B 0,C 180,E1 -917.906,E2 -917.906} C_VEL
LIN {X 0,Y 594.411,Z 214.442,A -85,B 0,C 180,E1 -920.775,E2 -920.775} C_VEL
LIN {X 0,Y 594.379,Z 214.45,A -85,B 0,C 180,E1 -923.705,E2 -923.705} C_VEL
LIN {X 0,Y 594.384,Z 214.444,A -85,B 0,C 180,E1 -926.021,E2 -926.021} C_VEL
LIN {X 0,Y 594.375,Z 214.451,A -85,B 0,C 180,E1 -928.999,E2 -928.999} C_VEL
LIN {X 0,Y 594.37,Z 214.444,A -85,B 0,C 180,E1 -931.641,E2 -931.641} C_VEL
LIN {X 0,Y 594.377,Z 214.451,A -85,B 0,C 180,E1 -934.137,E2 -934.137} C_VEL
LIN {X 0,Y 594.384,Z 214.445,A -85,B 0,C 180,E1 -937.087,E2 -937.087} C_VEL
LIN {X 0,Y 594.359,Z 214.447,A -85,B 0,C 180,E1 -939.772,E2 -939.772} C_VEL
LIN {X 0,Y 594.368,Z 214.449,A -85,B 0,C 180,E1 -942.376,E2 -942.376} C_VEL
LIN {X 0,Y 594.341,Z 214.448,A -85,B 0,C 180,E1 -945.194,E2 -945.194} C_VEL
LIN {X 0,Y 594.383,Z 214.445,A -85,B 0,C 180,E1 -948.152,E2 -948.152} C_VEL
LIN {X 0,Y 594.382,Z 214.451,A -85,B 0,C 180,E1 -951.194,E2 -951.194} C_VEL
LIN {X 0,Y 594.355,Z 214.447,A -85,B 0,C 180,E1 -953.755,E2 -953.755} C_VEL
LIN {X 0,Y 594.31,Z 214.46,A -85,B 0,C 180,E1 -954.683,E2 -954.683} C_VEL
LIN {X 0,Y 594.287,Z 217.035,A -85,B 0,C 180,E1 -957.103,E2 -957.103} C_VEL
LIN {X 0,Y 594.287,Z 219.981,A -85,B 0,C 180,E1 -959.689,E2 -959.689} C_VEL
LIN {X 0,Y 594.266,Z 223.289,A -85,B 0,C 180,E1 -962.533,E2 -962.533} C_VEL
LIN {X 0,Y 594.276,Z 226.937,A -85,B 0,C 180,E1 -965.591,E2 -965.591} C_VEL
LIN {X 0,Y 594.211,Z 230.726,A -85,B 0,C 180,E1 -968.491,E2 -968.491} C_VEL
LIN {X 0,Y 594.205,Z 233.609,A -85,B 0,C 180,E1 -970.66,E2 -970.66} C_VEL
LIN {X 0,Y 594.241,Z 237.452,A -85,B 0,C 180,E1 -973.51,E2 -973.51} C_VEL
LIN {X 0,Y 594.237,Z 241.295,A -85,B 0,C 180,E1 -976.317,E2 -976.317} C_VEL
LIN {X 0,Y 594.256,Z 243.668,A -85,B 0,C 180,E1 -978.034,E2 -978.034} C_VEL
LIN {X 0,Y 594.642,Z 248.439,A -85,B 0,C 180,E1 -978.15,E2 -978.15} C_VEL
LIN {X 0,Y 594.602,Z 261.032,A -85,B 0,C 180,E1 -978.492,E2 -978.492} C_VEL
LIN {X 0,Y 594.561,Z 272.839,A -85,B 0,C 180,E1 -978.942,E2 -978.942} C_VEL
LIN {X 0,Y 594.489,Z 284.522,A -85,B 0,C 180,E1 -979.527,E2 -979.527} C_VEL
LIN {X 0,Y 594.438,Z 295.313,A -85,B 0,C 180,E1 -980.215,E2 -980.215} C_VEL
LIN {X 0,Y 594.404,Z 305.089,A -85,B 0,C 180,E1 -980.987,E2 -980.987} C_VEL
LIN {X 0,Y 594.366,Z 313.984,A -85,B 0,C 180,E1 -981.842,E2 -981.842} C_VEL
LIN {X 0,Y 594.345,Z 322.67,A -85,B 0,C 180,E1 -982.868,E2 -982.868} C_VEL
LIN {X 0,Y 594.29,Z 329.599,A -85,B 0,C 180,E1 -983.89,E2 -983.89} C_VEL
LIN {X 0,Y 594.254,Z 335.151,A -85,B 0,C 180,E1 -984.911,E2 -984.911} C_VEL
LIN {X 0,Y 594.262,Z 339.513,A -85,B 0,C 180,E1 -985.931,E2 -985.931} C_VEL
LIN {X 0,Y 594.267,Z 341.816,A -85,B 0,C 180,E1 -986.61,E2 -986.61} C_VEL
LIN {X 0,Y 594.225,Z 343.694,A -85,B 0,C 180,E1 -987.288,E2 -987.288} C_VEL
LIN {X 0,Y 594.24,Z 345.127,A -85,B 0,C 180,E1 -987.967,E2 -987.967} C_VEL
LIN {X 0,Y 594.24,Z 346.753,A -85,B 0,C 180,E1 -989.322,E2 -989.322} C_VEL
LIN {X 0,Y 594.236,Z 346.996,A -85,B 0,C 180,E1 -990,E2 -990} C_VEL
LIN {X 0,Y 594.239,Z 346.815,A -85,B 0,C 180,E1 -990.678,E2 -990.678} C_VEL
LIN {X 0,Y 594.239,Z 345.275,A -85,B 0,C 180,E1 -992.033,E2 -992.033} C_VEL
LIN {X 0,Y 594.227,Z 343.915,A -85,B 0,C 180,E1 -992.712,E2 -992.712} C_VEL
LIN {X 0,Y 594.289,Z 341.038,A -85,B 0,C 180,E1 -993.729,E2 -993.729} C_VEL
LIN {X 0,Y 594.241,Z 337.139,A -85,B 0,C 180,E1 -994.749,E2 -994.749} C_VEL
LIN {X 0,Y 594.299,Z 332.107,A -85,B 0,C 180,E1 -995.769,E2 -995.769} C_VEL
LIN {X 0,Y 594.316,Z 325.788,A -85,B 0,C 180,E1 -996.791,E2 -996.791} C_VEL
LIN {X 0,Y 594.346,Z 317.87,A -85,B 0,C 180,E1 -997.816,E2 -997.816} C_VEL
LIN {X 0,Y 594.381,Z 308.024,A -85,B 0,C 180,E1 -998.842,E2 -998.842} C_VEL
LIN {X 0,Y 594.429,Z 297.703,A -85,B 0,C 180,E1 -999.699,E2 -999.699} C_VEL
LIN {X 0,Y 594.473,Z 287.497,A -85,B 0,C 180,E1 -1000.387,E2 -1000.387} C_VEL
LIN {X 0,Y 594.554,Z 275.673,A -85,B 0,C 180,E1 -1001.021,E2 -1001.021} C_VEL
LIN {X 0,Y 594.595,Z 263.559,A -85,B 0,C 180,E1 -1001.514,E2 -1001.514} C_VEL
LIN {X 0,Y 594.648,Z 250.428,A -85,B 0,C 180,E1 -1001.893,E2 -1001.893} C_VEL
LIN {X 0,Y 594.407,Z 245.034,A -85,B 0,C 180,E1 -1002.012,E2 -1002.012} C_VEL
LIN {X 0,Y 594.241,Z 243.643,A -85,B 0,C 180,E1 -1002.075,E2 -1002.075} C_VEL
LIN {X 0,Y 594.236,Z 240.458,A -85,B 0,C 180,E1 -1004.381,E2 -1004.381} C_VEL
LIN {X 0,Y 594.234,Z 236.613,A -85,B 0,C 180,E1 -1007.198,E2 -1007.198} C_VEL
LIN {X 0,Y 594.208,Z 233.729,A -85,B 0,C 180,E1 -1009.34,E2 -1009.34} C_VEL
LIN {X 0,Y 594.213,Z 230.845,A -85,B 0,C 180,E1 -1011.509,E2 -1011.509} C_VEL
LIN {X 0,Y 594.274,Z 227,A -85,B 0,C 180,E1 -1014.451,E2 -1014.451} C_VEL
LIN {X 0,Y 594.265,Z 223.366,A -85,B 0,C 180,E1 -1017.467,E2 -1017.467} C_VEL
LIN {X 0,Y 594.29,Z 220.11,A -85,B 0,C 180,E1 -1020.312,E2 -1020.312} C_VEL
LIN {X 0,Y 594.285,Z 217.094,A -85,B 0,C 180,E1 -1022.956,E2 -1022.956} C_VEL
LIN {X 0,Y 594.308,Z 214.46,A -85,B 0,C 180,E1 -1025.412,E2 -1025.412} C_VEL
LIN {X 0,Y 594.389,Z 214.442,A -85,B 0,C 180,E1 -1027.941,E2 -1027.941} C_VEL
LIN {X 0,Y 594.373,Z 214.449,A -85,B 0,C 180,E1 -1030.821,E2 -1030.821} C_VEL
LIN {X 0,Y 594.353,Z 214.447,A -85,B 0,C 180,E1 -1033.301,E2 -1033.301} C_VEL
LIN {X 0,Y 594.343,Z 214.45,A -85,B 0,C 180,E1 -1036.163,E2 -1036.163} C_VEL
LIN {X 0,Y 594.368,Z 214.445,A -85,B 0,C 180,E1 -1038.535,E2 -1038.535} C_VEL
LIN {X 0,Y 594.377,Z 214.446,A -85,B 0,C 180,E1 -1041.297,E2 -1041.297} C_VEL
LIN {X 0,Y 594.355,Z 214.448,A -85,B 0,C 180,E1 -1043.756,E2 -1043.756} C_VEL
LIN {X 0,Y 594.366,Z 214.449,A -85,B 0,C 180,E1 -1046.238,E2 -1046.238} C_VEL
LIN {X 0,Y 594.358,Z 214.446,A -85,B 0,C 180,E1 -1048.649,E2 -1048.649} C_VEL
LIN {X 0,Y 594.378,Z 214.45,A -85,B 0,C 180,E1 -1051.044,E2 -1051.044} C_VEL
LIN {X 0,Y 594.367,Z 214.447,A -85,B 0,C 180,E1 -1054.055,E2 -1054.055} C_VEL
LIN {X 0,Y 594.389,Z 214.45,A -85,B 0,C 180,E1 -1056.296,E2 -1056.296} C_VEL
LIN {X 0,Y 594.409,Z 214.442,A -85,B 0,C 180,E1 -1059.225,E2 -1059.225} C_VEL
LIN {X 0,Y 594.332,Z 214.449,A -85,B 0,C 180,E1 -1062.094,E2 -1062.094} C_VEL
LIN {X 0,Y 594.344,Z 214.448,A -85,B 0,C 180,E1 -1064.218,E2 -1064.218} C_VEL
LIN {X 0,Y 594.355,Z 214.448,A -85,B 0,C 180,E1 -1067.017,E2 -1067.017} C_VEL
LIN {X 0,Y 594.39,Z 214.448,A -85,B 0,C 180,E1 -1069.784,E2 -1069.784} C_VEL
LIN {X 0,Y 594.396,Z 214.441,A -85,B 0,C 180,E1 -1072.527,E2 -1072.527} C_VEL
LIN {X 0,Y 594.374,Z 214.449,A -85,B 0,C 180,E1 -1075.252,E2 -1075.252} C_VEL
LIN {X 0,Y 594.367,Z 214.446,A -85,B 0,C 180,E1 -1077.967,E2 -1077.967} C_VEL
LIN {X 0,Y 594.415,Z 214.44,A -85,B 0,C 180,E1 -1080.677,E2 -1080.677} C_VEL
LIN {X 0,Y 594.374,Z 214.449,A -85,B 0,C 180,E1 -1083.389,E2 -1083.389} C_VEL
LIN {X 0,Y 594.364,Z 214.445,A -85,B 0,C 180,E1 -1086.109,E2 -1086.109} C_VEL
LIN {X 0,Y 594.378,Z 214.449,A -85,B 0,C 180,E1 -1088.842,E2 -1088.842} C_VEL
LIN {X 0,Y 594.368,Z 214.446,A -85,B 0,C 180,E1 -1091.596,E2 -1091.596} C_VEL
LIN {X 0,Y 594.385,Z 214.444,A -85,B 0,C 180,E1 -1094.377,E2 -1094.377} C_VEL
LIN {X 0,Y 594.383,Z 214.45,A -85,B 0,C 180,E1 -1097.194,E2 -1097.194} C_VEL
LIN {X 0,Y 594.377,Z 214.444,A -85,B 0,C 180,E1 -1100.054,E2 -1100.054} C_VEL
LIN {X 0,Y 594.356,Z 214.447,A -85,B 0,C 180,E1 -1102.968,E2 -1102.968} C_VEL
LIN {X 0,Y 594.333,Z 214.45,A -85,B 0,C 180,E1 -1105.195,E2 -1105.195} C_VEL
LIN {X 0,Y 594.345,Z 214.456,A -85,B 0,C 180,E1 -1107.518,E2 -1107.518} C_VEL
LIN {X 0,Y 594.371,Z 214.445,A -85,B 0,C 180,E1 -1110.325,E2 -1110.325} C_VEL
LIN {X 0,Y 594.382,Z 214.446,A -85,B 0,C 180,E1 -1112.95,E2 -1112.95} C_VEL
LIN {X 0,Y 594.351,Z 214.447,A -85,B 0,C 180,E1 -1115.409,E2 -1115.409} C_VEL
LIN {X 0,Y 594.372,Z 214.449,A -85,B 0,C 180,E1 -1117.942,E2 -1117.942} C_VEL
LIN {X 0,Y 594.36,Z 214.448,A -85,B 0,C 180,E1 -1120.82,E2 -1120.82} C_VEL
LIN {X 0,Y 594.362,Z 214.446,A -85,B 0,C 180,E1 -1123.839,E2 -1123.839} C_VEL
LIN {X 0,Y 594.368,Z 214.447,A -85,B 0,C 180,E1 -1126.7,E2 -1126.7} C_VEL
LIN {X 0,Y 594.369,Z 214.449,A -85,B 0,C 180,E1 -1129.433,E2 -1129.433} C_VEL
LIN {X 0,Y 594.383,Z 214.444,A -85,B 0,C 180,E1 -1132.393,E2 -1132.393} C_VEL
LIN {X 0,Y 594.38,Z 214.635,A -85,B 0,C 180,E1 -1133.967,E2 -1133.967} C_VEL
LIN {X 0,Y 594.615,Z 219.268,A -85,B 0,C 180,E1 -1135.435,E2 -1135.435} C_VEL
LIN {X 0,Y 594.567,Z 227.212,A -85,B 0,C 180,E1 -1137.865,E2 -1137.865} C_VEL
LIN {X 0,Y 594.564,Z 236.479,A -85,B 0,C 180,E1 -1140.623,E2 -1140.623} C_VEL
LIN {X 0,Y 594.47,Z 245.746,A -85,B 0,C 180,E1 -1143.305,E2 -1143.305} C_VEL
LIN {X 0,Y 594.446,Z 255.014,A -85,B 0,C 180,E1 -1145.928,E2 -1145.928} C_VEL
LIN {X 0,Y 594.404,Z 265.493,A -85,B 0,C 180,E1 -1148.831,E2 -1148.831} C_VEL
LIN {X 0,Y 594.375,Z 274.872,A -85,B 0,C 180,E1 -1151.382,E2 -1151.382} C_VEL
LIN {X 0,Y 594.318,Z 285.464,A -85,B 0,C 180,E1 -1154.218,E2 -1154.218} C_VEL
LIN {X 0,Y 594.275,Z 296.055,A -85,B 0,C 180,E1 -1157.015,E2 -1157.015} C_VEL
LIN {X 0,Y 594.283,Z 299.53,A -85,B 0,C 180,E1 -1157.926,E2 -1157.926} C_VEL
LIN {X 0,Y 594.668,Z 305.231,A -85,B 0,C 180,E1 -1158.042,E2 -1158.042} C_VEL
LIN {X 0,Y 594.614,Z 318.496,A -85,B 0,C 180,E1 -1158.365,E2 -1158.365} C_VEL
LIN {X 0,Y 594.529,Z 330.658,A -85,B 0,C 180,E1 -1158.802,E2 -1158.802} C_VEL
LIN {X 0,Y 594.472,Z 342.208,A -85,B 0,C 180,E1 -1159.355,E2 -1159.355} C_VEL
LIN {X 0,Y 594.459,Z 353.476,A -85,B 0,C 180,E1 -1160.043,E2 -1160.043} C_VEL
LIN {X 0,Y 594.406,Z 363.647,A -85,B 0,C 180,E1 -1160.815,E2 -1160.815} C_VEL
LIN {X 0,Y 594.372,Z 372.788,A -85,B 0,C 180,E1 -1161.672,E2 -1161.672} C_VEL
LIN {X 0,Y 594.316,Z 381.691,A -85,B 0,C 180,E1 -1162.697,E2 -1162.697} C_VEL
LIN {X 0,Y 594.281,Z 388.169,A -85,B 0,C 180,E1 -1163.615,E2 -1163.615} C_VEL
LIN {X 0,Y 594.289,Z 393.68,A -85,B 0,C 180,E1 -1164.571,E2 -1164.571} C_VEL
LIN {X 0,Y 594.27,Z 398.371,A -85,B 0,C 180,E1 -1165.591,E2 -1165.591} C_VEL
LIN {X 0,Y 594.267,Z 401.956,A -85,B 0,C 180,E1 -1166.61,E2 -1166.61} C_VEL
LIN {X 0,Y 594.226,Z 403.809,A -85,B 0,C 180,E1 -1167.288,E2 -1167.288} C_VEL
LIN {X 0,Y 594.242,Z 405.202,A -85,B 0,C 180,E1 -1167.967,E2 -1167.967} C_VEL
LIN {X 0,Y 594.239,Z 406.784,A -85,B 0,C 180,E1 -1169.322,E2 -1169.322} C_VEL
LIN {X 0,Y 594.236,Z 407,A -85,B 0,C 180,E1 -1170,E2 -1170} C_VEL
LIN {X 0,Y 594.247,Z 406.184,A -85,B 0,C 180,E1 -1171.355,E2 -1171.355} C_VEL
LIN {X 0,Y 594.242,Z 405.202,A -85,B 0,C 180,E1 -1172.033,E2 -1172.033} C_VEL
LIN {X 0,Y 594.226,Z 403.809,A -85,B 0,C 180,E1 -1172.712,E2 -1172.712} C_VEL
LIN {X 0,Y 594.289,Z 400.896,A -85,B 0,C 180,E1 -1173.729,E2 -1173.729} C_VEL
LIN {X 0,Y 594.241,Z 396.949,A -85,B 0,C 180,E1 -1174.749,E2 -1174.749} C_VEL
LIN {X 0,Y 594.305,Z 390.876,A -85,B 0,C 180,E1 -1175.939,E2 -1175.939} C_VEL
LIN {X 0,Y 594.308,Z 384.234,A -85,B 0,C 180,E1 -1176.962,E2 -1176.962} C_VEL
LIN {X 0,Y 594.359,Z 375.988,A -85,B 0,C 180,E1 -1177.987,E2 -1177.987} C_VEL
LIN {X 0,Y 594.382,Z 367.535,A -85,B 0,C 180,E1 -1178.842,E2 -1178.842} C_VEL
LIN {X 0,Y 594.432,Z 357.09,A -85,B 0,C 180,E1 -1179.7,E2 -1179.7} C_VEL
LIN {X 0,Y 594.45,Z 346.754,A -85,B 0,C 180,E1 -1180.387,E2 -1180.387} C_VEL
LIN {X 0,Y 594.499,Z 334.775,A -85,B 0,C 180,E1 -1181.019,E2 -1181.019} C_VEL
LIN {X 0,Y 594.56,Z 322.489,A -85,B 0,C 180,E1 -1181.505,E2 -1181.505} C_VEL
LIN {X 0,Y 594.673,Z 309.43,A -85,B 0,C 180,E1 -1181.871,E2 -1181.871} C_VEL
LIN {X 0,Y 594.453,Z 300.849,A -85,B 0,C 180,E1 -1182.038,E2 -1182.038} C_VEL
LIN {X 0,Y 594.283,Z 299.53,A -85,B 0,C 180,E1 -1182.074,E2 -1182.074} C_VEL
LIN {X 0,Y 594.305,Z 289.435,A -85,B 0,C 180,E1 -1184.729,E2 -1184.729} C_VEL
LIN {X 0,Y 594.336,Z 278.843,A -85,B 0,C 180,E1 -1187.55,E2 -1187.55} C_VEL
LIN {X 0,Y 594.383,Z 268.252,A -85,B 0,C 180,E1 -1190.415,E2 -1190.415} C_VEL
LIN {X 0,Y 594.441,Z 257.661,A -85,B 0,C 180,E1 -1193.333,E2 -1193.333} C_VEL
LIN {X 0,Y 594.488,Z 248.031,A -85,B 0,C 180,E1 -1196.042,E2 -1196.042} C_VEL
LIN {X 0,Y 594.487,Z 239.147,A -85,B 0,C 180,E1 -1198.601,E2 -1198.601} C_VEL
LIN {X 0,Y 594.588,Z 229.859,A -85,B 0,C 180,E1 -1201.338,E2 -1201.338} C_VEL
LIN {X 0,Y 594.613,Z 221.915,A -85,B 0,C 180,E1 -1203.747,E2 -1203.747} C_VEL
LIN {X 0,Y 594.495,Z 215.296,A -85,B 0,C 180,E1 -1205.816,E2 -1205.816} C_VEL
LIN {X 0,Y 594.359,Z 214.452,A -85,B 0,C 180,E1 -1206.139,E2 -1206.139} C_VEL
LIN {X 0,Y 594.369,Z 214.45,A -85,B 0,C 180,E1 -1208.807,E2 -1208.807} C_VEL
LIN {X 0,Y 594.385,Z 214.449,A -85,B 0,C 180,E1 -1211.848,E2 -1211.848} C_VEL
LIN {X 0,Y 594.364,Z 214.447,A -85,B 0,C 180,E1 -1214.239,E2 -1214.239} C_VEL
LIN {X 0,Y 594.364,Z 214.447,A -85,B 0,C 180,E1 -1216.7,E2 -1216.7} C_VEL
LIN {X 0,Y 594.342,Z 214.448,A -85,B 0,C 180,E1 -1219.431,E2 -1219.431} C_VEL
LIN {X 0,Y 594.381,Z 214.449,A -85,B 0,C 180,E1 -1222.393,E2 -1222.393} C_VEL
LIN {X 0,Y 594.376,Z 214.448,A -85,B 0,C 180,E1 -1225.42,E2 -1225.42} C_VEL
LIN {X 0,Y 594.381,Z 214.443,A -85,B 0,C 180,E1 -1228.358,E2 -1228.358} C_VEL
LIN {X 0,Y 594.378,Z 214.448,A -85,B 0,C 180,E1 -1231.044,E2 -1231.044} C_VEL
LIN {X 0,Y 594.362,Z 214.451,A -85,B 0,C 180,E1 -1234.055,E2 -1234.055} C_VEL
LIN {X 0,Y 594.365,Z 214.448,A -85,B 0,C 180,E1 -1236.295,E2 -1236.295} C_VEL
LIN {X 0,Y 594.407,Z 214.446,A -85,B 0,C 180,E1 -1239.224,E2 -1239.224} C_VEL
LIN {X 0,Y 594.359,Z 214.446,A -85,B 0,C 180,E1 -1242.095,E2 -1242.095} C_VEL
LIN {X 0,Y 594.363,Z 214.449,A -85,B 0,C 180,E1 -1244.219,E2 -1244.219} C_VEL
LIN {X 0,Y 594.371,Z 214.45,A -85,B 0,C 180,E1 -1246.321,E2 -1246.321} C_VEL
LIN {X 0,Y 594.327,Z 214.451,A -85,B 0,C 180,E1 -1249.094,E2 -1249.094} C_VEL
LIN {X 0,Y 594.365,Z 214.446,A -85,B 0,C 180,E1 -1251.843,E2 -1251.843} C_VEL
LIN {X 0,Y 594.397,Z 214.447,A -85,B 0,C 180,E1 -1254.572,E2 -1254.572} C_VEL
LIN {X 0,Y 594.408,Z 214.44,A -85,B 0,C 180,E1 -1257.289,E2 -1257.289} C_VEL
LIN {X 0,Y 594.409,Z 214.446,A -85,B 0,C 180,E1 -1260,E2 -1260} C_VEL
LIN {X 0,Y 594.375,Z 214.444,A -85,B 0,C 180,E1 -1262.711,E2 -1262.711} C_VEL
LIN {X 0,Y 594.394,Z 214.444,A -85,B 0,C 180,E1 -1265.428,E2 -1265.428} C_VEL
LIN {X 0,Y 594.367,Z 214.449,A -85,B 0,C 180,E1 -1268.157,E2 -1268.157} C_VEL
LIN {X 0,Y 594.39,Z 214.442,A -85,B 0,C 180,E1 -1271.071,E2 -1271.071} C_VEL
LIN {X 0,Y 594.366,Z 214.451,A -85,B 0,C 180,E1 -1273.679,E2 -1273.679} C_VEL
LIN {X 0,Y 594.336,Z 214.451,A -85,B 0,C 180,E1 -1275.314,E2 -1275.314} C_VEL
LIN {X 0,Y 593.661,Z 214.535,A -85,B 0,C 180,E1 -1275.88,E2 -1275.88} C_VEL
LIN {X 0,Y 590.792,Z 214.895,A -85,B 0,C 180,E1 -1276.797,E2 -1276.797} C_VEL
LIN {X 0,Y 588.383,Z 215.193,A -85,B 0,C 180,E1 -1277.535,E2 -1277.535} C_VEL
LIN {X 0,Y 587.367,Z 215.318,A -85,B 0,C 180,E1 -1278.105,E2 -1278.105} C_VEL
LIN {X 0,Y 587.294,Z 215.327,A -85,B 0,C 180,E1 -1278.298,E2 -1278.298} C_VEL
LIN {X 0,Y 587.337,Z 215.321,A -85,B 0,C 180,E1 -1281.037,E2 -1281.037} C_VEL
LIN {X 0,Y 587.319,Z 215.324,A -85,B 0,C 180,E1 -1283.259,E2 -1283.259} C_VEL
LIN {X 0,Y 587.336,Z 215.328,A -85,B 0,C 180,E1 -1285.517,E2 -1285.517} C_VEL
LIN {X 0,Y 587.297,Z 215.326,A -85,B 0,C 180,E1 -1287.82,E2 -1287.82} C_VEL
LIN {X 0,Y 587.295,Z 215.327,A -85,B 0,C 180,E1 -1290.173,E2 -1290.173} C_VEL
LIN {X 0,Y 587.341,Z 215.325,A -85,B 0,C 180,E1 -1292.579,E2 -1292.579} C_VEL
LIN {X 0,Y 587.326,Z 215.322,A -85,B 0,C 180,E1 -1295.056,E2 -1295.056} C_VEL
LIN {X 0,Y 587.341,Z 215.323,A -85,B 0,C 180,E1 -1297.838,E2 -1297.838} C_VEL
LIN {X 0,Y 587.313,Z 215.324,A -85,B 0,C 180,E1 -1300.255,E2 -1300.255} C_VEL
LIN {X 0,Y 587.305,Z 215.327,A -85,B 0,C 180,E1 -1303.008,E2 -1303.008} C_VEL
LIN {X 0,Y 587.303,Z 215.333,A -85,B 0,C 180,E1 -1306.047,E2 -1306.047} C_VEL
LIN {X 0,Y 587.335,Z 215.322,A -85,B 0,C 180,E1 -1308.926,E2 -1308.926} C_VEL
LIN {X 0,Y 587.333,Z 215.324,A -85,B 0,C 180,E1 -1311.52,E2 -1311.52} C_VEL
LIN {X 0,Y 587.282,Z 215.329,A -85,B 0,C 180,E1 -1314.099,E2 -1314.099} C_VEL
LIN {X 0,Y 587.224,Z 215.342,A -85,B 0,C 180,E1 -1314.937,E2 -1314.937} C_VEL
LIN {X 0,Y 587.2,Z 218.072,A -85,B 0,C 180,E1 -1317.412,E2 -1317.412} C_VEL
LIN {X 0,Y 587.226,Z 220.767,A -85,B 0,C 180,E1 -1319.823,E2 -1319.823} C_VEL
LIN {X 0,Y 587.201,Z 223.64,A -85,B 0,C 180,E1 -1322.336,E2 -1322.336} C_VEL
LIN {X 0,Y 587.168,Z 226.985,A -85,B 0,C 180,E1 -1325.233,E2 -1325.233} C_VEL
LIN {X 0,Y 587.151,Z 229.766,A -85,B 0,C 180,E1 -1327.478,E2 -1327.478} C_VEL
LIN {X 0,Y 587.162,Z 232.649,A -85,B 0,C 180,E1 -1329.689,E2 -1329.689} C_VEL
LIN {X 0,Y 587.121,Z 235.531,A -85,B 0,C 180,E1 -1331.867,E2 -1331.867} C_VEL
LIN {X 0,Y 587.147,Z 238.414,A -85,B 0,C 180,E1 -1334.02,E2 -1334.02} C_VEL
LIN {X 0,Y 587.136,Z 242.257,A -85,B 0,C 180,E1 -1336.854,E2 -1336.854} C_VEL
LIN {X 0,Y 587.136,Z 243.668,A -85,B 0,C 180,E1 -1337.886,E2 -1337.886} C_VEL
LIN {X 0,Y 587.697,Z 249.376,A -85,B 0,C 180,E1 -1338.029,E2 -1338.029} C_VEL
LIN {X 0,Y 587.63,Z 262.589,A -85,B 0,C 180,E1 -1338.405,E2 -1338.405} C_VEL
LIN {X 0,Y 587.599,Z 274.628,A -85,B 0,C 180,E1 -1338.888,E2 -1338.888} C_VEL
LIN {X 0,Y 587.481,Z 286.018,A -85,B 0,C 180,E1 -1339.488,E2 -1339.488} C_VEL
LIN {X 0,Y 587.421,Z 297.654,A -85,B 0,C 180,E1 -1340.271,E2 -1340.271} C_VEL
LIN {X 0,Y 587.344,Z 307.035,A -85,B 0,C 180,E1 -1341.051,E2 -1341.051} C_VEL
LIN {X 0,Y 587.3,Z 315.599,A -85,B 0,C 180,E1 -1341.917,E2 -1341.917} C_VEL
LIN {X 0,Y 587.262,Z 323.914,A -85,B 0,C 180,E1 -1342.954,E2 -1342.954} C_VEL
LIN {X 0,Y 587.218,Z 330.613,A -85,B 0,C 180,E1 -1343.989,E2 -1343.989} C_VEL
LIN {X 0,Y 587.146,Z 336.757,A -85,B 0,C 180,E1 -1345.194,E2 -1345.194} C_VEL
LIN {X 0,Y 587.212,Z 340.747,A -85,B 0,C 180,E1 -1346.226,E2 -1346.226} C_VEL
LIN {X 0,Y 587.131,Z 343.696,A -85,B 0,C 180,E1 -1347.255,E2 -1347.255} C_VEL
LIN {X 0,Y 587.139,Z 345.127,A -85,B 0,C 180,E1 -1347.942,E2 -1347.942} C_VEL
LIN {X 0,Y 587.14,Z 346.754,A -85,B 0,C 180,E1 -1349.314,E2 -1349.314} C_VEL
LIN {X 0,Y 587.137,Z 346.996,A -85,B 0,C 180,E1 -1350,E2 -1350} C_VEL
LIN {X 0,Y 587.14,Z 346.815,A -85,B 0,C 180,E1 -1350.686,E2 -1350.686} C_VEL
LIN {X 0,Y 587.138,Z 345.274,A -85,B 0,C 180,E1 -1352.058,E2 -1352.058} C_VEL
LIN {X 0,Y 587.133,Z 343.913,A -85,B 0,C 180,E1 -1352.744,E2 -1352.744} C_VEL
LIN {X 0,Y 587.213,Z 341.036,A -85,B 0,C 180,E1 -1353.774,E2 -1353.774} C_VEL
LIN {X 0,Y 587.147,Z 337.136,A -85,B 0,C 180,E1 -1354.806,E2 -1354.806} C_VEL
LIN {X 0,Y 587.229,Z 332.105,A -85,B 0,C 180,E1 -1355.839,E2 -1355.839} C_VEL
LIN {X 0,Y 587.23,Z 325.784,A -85,B 0,C 180,E1 -1356.874,E2 -1356.874} C_VEL
LIN {X 0,Y 587.288,Z 317.865,A -85,B 0,C 180,E1 -1357.91,E2 -1357.91} C_VEL
LIN {X 0,Y 587.343,Z 308.018,A -85,B 0,C 180,E1 -1358.949,E2 -1358.949} C_VEL
LIN {X 0,Y 587.411,Z 297.697,A -85,B 0,C 180,E1 -1359.816,E2 -1359.816} C_VEL
LIN {X 0,Y 587.496,Z 286.067,A -85,B 0,C 180,E1 -1360.598,E2 -1360.598} C_VEL
LIN {X 0,Y 587.568,Z 275.125,A -85,B 0,C 180,E1 -1361.179,E2 -1361.179} C_VEL
LIN {X 0,Y 587.624,Z 262.456,A -85,B 0,C 180,E1 -1361.689,E2 -1361.689} C_VEL
LIN {X 0,Y 587.704,Z 249.49,A -85,B 0,C 180,E1 -1362.058,E2 -1362.058} C_VEL
LIN {X 0,Y 587.374,Z 245.29,A -85,B 0,C 180,E1 -1362.152,E2 -1362.152} C_VEL
LIN {X 0,Y 587.142,Z 243.672,A -85,B 0,C 180,E1 -1362.201,E2 -1362.201} C_VEL
LIN {X 0,Y 587.129,Z 240.458,A -85,B 0,C 180,E1 -1364.559,E2 -1364.559} C_VEL
LIN {X 0,Y 587.147,Z 237.503,A -85,B 0,C 180,E1 -1366.747,E2 -1366.747} C_VEL
LIN {X 0,Y 587.113,Z 233.728,A -85,B 0,C 180,E1 -1369.583,E2 -1369.583} C_VEL
LIN {X 0,Y 587.132,Z 230.844,A -85,B 0,C 180,E1 -1371.782,E2 -1371.782} C_VEL
LIN {X 0,Y 587.191,Z 227.358,A -85,B 0,C 180,E1 -1374.545,E2 -1374.545} C_VEL
LIN {X 0,Y 587.168,Z 224.465,A -85,B 0,C 180,E1 -1377.054,E2 -1377.054} C_VEL
LIN {X 0,Y 587.202,Z 221.807,A -85,B 0,C 180,E1 -1379.388,E2 -1379.388} C_VEL
LIN {X 0,Y 587.201,Z 219.057,A -85,B 0,C 180,E1 -1381.813,E2 -1381.813} C_VEL
LIN {X 0,Y 587.256,Z 216.233,A -85,B 0,C 180,E1 -1384.334,E2 -1384.334} C_VEL
LIN {X 0,Y 587.219,Z 215.397,A -85,B 0,C 180,E1 -1385.063,E2 -1385.063} C_VEL
LIN {X 0,Y 587.348,Z 215.322,A -85,B 0,C 180,E1 -1387.608,E2 -1387.608} C_VEL
LIN {X 0,Y 587.315,Z 215.326,A -85,B 0,C 180,E1 -1390.254,E2 -1390.254} C_VEL
LIN {X 0,Y 587.305,Z 215.325,A -85,B 0,C 180,E1 -1393.117,E2 -1393.117} C_VEL
LIN {X 0,Y 587.299,Z 215.329,A -85,B 0,C 180,E1 -1396.047,E2 -1396.047} C_VEL
LIN {X 0,Y 587.332,Z 215.326,A -85,B 0,C 180,E1 -1398.926,E2 -1398.926} C_VEL
LIN {X 0,Y 587.326,Z 215.323,A -85,B 0,C 180,E1 -1401.52,E2 -1401.52} C_VEL
LIN {X 0,Y 587.295,Z 215.331,A -85,B 0,C 180,E1 -1404.1,E2 -1404.1} C_VEL
LIN {X 0,Y 587.339,Z 215.32,A -85,B 0,C 180,E1 -1406.889,E2 -1406.889} C_VEL
LIN {X 0,Y 587.306,Z 215.331,A -85,B 0,C 180,E1 -1409.496,E2 -1409.496} C_VEL
LIN {X 0,Y 587.302,Z 215.329,A -85,B 0,C 180,E1 -1411.402,E2 -1411.402} C_VEL
LIN {X 0,Y 587.34,Z 215.321,A -85,B 0,C 180,E1 -1413.824,E2 -1413.824} C_VEL
LIN {X 0,Y 587.329,Z 215.326,A -85,B 0,C 180,E1 -1415.993,E2 -1415.993} C_VEL
LIN {X 0,Y 587.324,Z 215.326,A -85,B 0,C 180,E1 -1418.226,E2 -1418.226} C_VEL
LIN {X 0,Y 587.349,Z 215.323,A -85,B 0,C 180,E1 -1421.151,E2 -1421.151} C_VEL
LIN {X 0,Y 587.299,Z 215.325,A -85,B 0,C 180,E1 -1424.024,E2 -1424.024} C_VEL
LIN {X 0,Y 587.305,Z 215.328,A -85,B 0,C 180,E1 -1426.858,E2 -1426.858} C_VEL
LIN {X 0,Y 587.34,Z 215.325,A -85,B 0,C 180,E1 -1429.66,E2 -1429.66} C_VEL
LIN {X 0,Y 587.366,Z 215.317,A -85,B 0,C 180,E1 -1432.437,E2 -1432.437} C_VEL
LIN {X 0,Y 587.348,Z 215.325,A -85,B 0,C 180,E1 -1435.195,E2 -1435.195} C_VEL
LIN {X 0,Y 587.34,Z 215.321,A -85,B 0,C 180,E1 -1437.943,E2 -1437.943} C_VEL
LIN {X 0,Y 587.387,Z 215.316,A -85,B 0,C 180,E1 -1440.686,E2 -1440.686} C_VEL
LIN {X 0,Y 587.327,Z 215.328,A -85,B 0,C 180,E1 -1443.43,E2 -1443.43} C_VEL
LIN {X 0,Y 587.361,Z 215.323,A -85,B 0,C 180,E1 -1445.493,E2 -1445.493} C_VEL
LIN {X 0,Y 587.33,Z 215.323,A -85,B 0,C 180,E1 -1448.256,E2 -1448.256} C_VEL
LIN {X 0,Y 587.3,Z 215.325,A -85,B 0,C 180,E1 -1451.107,E2 -1451.107} C_VEL
LIN {X 0,Y 587.343,Z 215.322,A -85,B 0,C 180,E1 -1454.25,E2 -1454.25} C_VEL
LIN {X 0,Y 587.349,Z 215.325,A -85,B 0,C 180,E1 -1457.406,E2 -1457.406} C_VEL
LIN {X 0,Y 587.332,Z 215.324,A -85,B 0,C 180,E1 -1460.305,E2 -1460.305} C_VEL
LIN {X 0,Y 587.311,Z 215.324,A -85,B 0,C 180,E1 -1463.259,E2 -1463.259} C_VEL
LIN {X 0,Y 587.306,Z 215.327,A -85,B 0,C 180,E1 -1466.17,E2 -1466.17} C_VEL
LIN {X 0,Y 587.345,Z 215.326,A -85,B 0,C 180,E1 -1469.132,E2 -1469.132} C_VEL
LIN {X 0,Y 587.352,Z 215.319,A -85,B 0,C 180,E1 -1471.836,E2 -1471.836} C_VEL
LIN {X 0,Y 587.347,Z 215.327,A -85,B 0,C 180,E1 -1474.347,E2 -1474.347} C_VEL
LIN {X 0,Y 587.34,Z 215.326,A -85,B 0,C 180,E1 -1477.608,E2 -1477.608} C_VEL
LIN {X 0,Y 587.292,Z 215.326,A -85,B 0,C 180,E1 -1480.256,E2 -1480.256} C_VEL
LIN {X 0,Y 587.306,Z 215.329,A -85,B 0,C 180,E1 -1483.117,E2 -1483.117} C_VEL
LIN {X 0,Y 587.315,Z 215.328,A -85,B 0,C 180,E1 -1486.048,E2 -1486.048} C_VEL
LIN {X 0,Y 587.337,Z 215.321,A -85,B 0,C 180,E1 -1488.925,E2 -1488.925} C_VEL
LIN {X 0,Y 587.318,Z 215.331,A -85,B 0,C 180,E1 -1491.52,E2 -1491.52} C_VEL
LIN {X 0,Y 587.337,Z 215.462,A -85,B 0,C 180,E1 -1493.732,E2 -1493.732} C_VEL
LIN {X 0,Y 587.66,Z 220.417,A -85,B 0,C 180,E1 -1495.329,E2 -1495.329} C_VEL
LIN {X 0,Y 587.619,Z 228.457,A -85,B 0,C 180,E1 -1497.82,E2 -1497.82} C_VEL
LIN {X 0,Y 587.569,Z 237.803,A -85,B 0,C 180,E1 -1500.633,E2 -1500.633} C_VEL
LIN {X 0,Y 587.477,Z 247.07,A -85,B 0,C 180,E1 -1503.345,E2 -1503.345} C_VEL
LIN {X 0,Y 587.42,Z 256.338,A -85,B 0,C 180,E1 -1505.997,E2 -1505.997} C_VEL
LIN {X 0,Y 587.359,Z 265.606,A -85,B 0,C 180,E1 -1508.596,E2 -1508.596} C_VEL
LIN {X 0,Y 587.32,Z 276.196,A -85,B 0,C 180,E1 -1511.512,E2 -1511.512} C_VEL
LIN {X 0,Y 587.258,Z 286.788,A -85,B 0,C 180,E1 -1514.379,E2 -1514.379} C_VEL
LIN {X 0,Y 587.202,Z 297.379,A -85,B 0,C 180,E1 -1517.208,E2 -1517.208} C_VEL
LIN {X 0,Y 587.195,Z 299.572,A -85,B 0,C 180,E1 -1517.789,E2 -1517.789} C_VEL
LIN {X 0,Y 587.738,Z 304.089,A -85,B 0,C 180,E1 -1517.877,E2 -1517.877} C_VEL
LIN {X 0,Y 587.671,Z 317.737,A -85,B 0,C 180,E1 -1518.204,E2 -1518.204} C_VEL
LIN {X 0,Y 587.563,Z 330.435,A -85,B 0,C 180,E1 -1518.657,E2 -1518.657} C_VEL
LIN {X 0,Y 587.49,Z 342.209,A -85,B 0,C 180,E1 -1519.227,E2 -1519.227} C_VEL
LIN {X 0,Y 587.456,Z 353.477,A -85,B 0,C 180,E1 -1519.923,E2 -1519.923} C_VEL
LIN {X 0,Y 587.384,Z 363.647,A -85,B 0,C 180,E1 -1520.705,E2 -1520.705} C_VEL
LIN {X 0,Y 587.34,Z 372.788,A -85,B 0,C 180,E1 -1521.571,E2 -1521.571} C_VEL
LIN {X 0,Y 587.259,Z 381.691,A -85,B 0,C 180,E1 -1522.608,E2 -1522.608} C_VEL
LIN {X 0,Y 587.195,Z 388.746,A -85,B 0,C 180,E1 -1523.627,E2 -1523.627} C_VEL
LIN {X 0,Y 587.211,Z 393.681,A -85,B 0,C 180,E1 -1524.506,E2 -1524.506} C_VEL
LIN {X 0,Y 587.188,Z 398.371,A -85,B 0,C 180,E1 -1525.538,E2 -1525.538} C_VEL
LIN {X 0,Y 587.193,Z 401.956,A -85,B 0,C 180,E1 -1526.569,E2 -1526.569} C_VEL
LIN {X 0,Y 587.132,Z 403.809,A -85,B 0,C 180,E1 -1527.256,E2 -1527.256} C_VEL
LIN {X 0,Y 587.141,Z 405.202,A -85,B 0,C 180,E1 -1527.942,E2 -1527.942} C_VEL
LIN {X 0,Y 587.14,Z 406.784,A -85,B 0,C 180,E1 -1529.314,E2 -1529.314} C_VEL
LIN {X 0,Y 587.137,Z 407,A -85,B 0,C 180,E1 -1530,E2 -1530} C_VEL
LIN {X 0,Y 587.147,Z 406.184,A -85,B 0,C 180,E1 -1531.372,E2 -1531.372} C_VEL
LIN {X 0,Y 587.141,Z 405.202,A -85,B 0,C 180,E1 -1532.058,E2 -1532.058} C_VEL
LIN {X 0,Y 587.132,Z 403.809,A -85,B 0,C 180,E1 -1532.745,E2 -1532.745} C_VEL
LIN {X 0,Y 587.213,Z 400.896,A -85,B 0,C 180,E1 -1533.774,E2 -1533.774} C_VEL
LIN {X 0,Y 587.147,Z 396.949,A -85,B 0,C 180,E1 -1534.806,E2 -1534.806} C_VEL
LIN {X 0,Y 587.218,Z 390.876,A -85,B 0,C 180,E1 -1536.011,E2 -1536.011} C_VEL
LIN {X 0,Y 587.245,Z 384.235,A -85,B 0,C 180,E1 -1537.046,E2 -1537.046} C_VEL
LIN {X 0,Y 587.299,Z 375.988,A -85,B 0,C 180,E1 -1538.083,E2 -1538.083} C_VEL
LIN {X 0,Y 587.343,Z 367.535,A -85,B 0,C 180,E1 -1538.949,E2 -1538.949} C_VEL
LIN {X 0,Y 587.415,Z 357.09,A -85,B 0,C 180,E1 -1539.817,E2 -1539.817} C_VEL
LIN {X 0,Y 587.451,Z 346.755,A -85,B 0,C 180,E1 -1540.512,E2 -1540.512} C_VEL
LIN {X 0,Y 587.529,Z 335.166,A -85,B 0,C 180,E1 -1541.133,E2 -1541.133} C_VEL
LIN {X 0,Y 587.594,Z 322.692,A -85,B 0,C 180,E1 -1541.637,E2 -1541.637} C_VEL
LIN {X 0,Y 587.72,Z 309.43,A -85,B 0,C 180,E1 -1542.014,E2 -1542.014} C_VEL
LIN {X 0,Y 587.489,Z 301.6,A -85,B 0,C 180,E1 -1542.172,E2 -1542.172} C_VEL
LIN {X 0,Y 587.193,Z 299.53,A -85,B 0,C 180,E1 -1542.222,E2 -1542.222} C_VEL
LIN {X 0,Y 587.255,Z 289.435,A -85,B 0,C 180,E1 -1544.91,E2 -1544.91} C_VEL
LIN {X 0,Y 587.298,Z 278.843,A -85,B 0,C 180,E1 -1547.767,E2 -1547.767} C_VEL
LIN {X 0,Y 587.378,Z 268.252,A -85,B 0,C 180,E1 -1550.669,E2 -1550.669} C_VEL
LIN {X 0,Y 587.436,Z 257.661,A -85,B 0,C 180,E1 -1553.628,E2 -1553.628} C_VEL
LIN {X 0,Y 587.49,Z 248.394,A -85,B 0,C 180,E1 -1556.272,E2 -1556.272} C_VEL
LIN {X 0,Y 587.491,Z 240.45,A -85,B 0,C 180,E1 -1558.588,E2 -1558.588} C_VEL
LIN {X 0,Y 587.619,Z 231.183,A -85,B 0,C 180,E1 -1561.35,E2 -1561.35} C_VEL
LIN {X 0,Y 587.65,Z 223.239,A -85,B 0,C 180,E1 -1563.788,E2 -1563.788} C_VEL
LIN {X 0,Y 587.539,Z 216.62,A -85,B 0,C 180,E1 -1565.883,E2 -1565.883} C_VEL
LIN {X 0,Y 587.305,Z 215.331,A -85,B 0,C 180,E1 -1566.324,E2 -1566.324} C_VEL
LIN {X 0,Y 587.315,Z 215.327,A -85,B 0,C 180,E1 -1568.939,E2 -1568.939} C_VEL
LIN {X 0,Y 587.338,Z 215.321,A -85,B 0,C 180,E1 -1571.157,E2 -1571.157} C_VEL
LIN {X 0,Y 587.316,Z 215.326,A -85,B 0,C 180,E1 -1574.112,E2 -1574.112} C_VEL
LIN {X 0,Y 587.303,Z 215.331,A -85,B 0,C 180,E1 -1576.992,E2 -1576.992} C_VEL
LIN {X 0,Y 587.294,Z 215.326,A -85,B 0,C 180,E1 -1579.744,E2 -1579.744} C_VEL
LIN {X 0,Y 587.336,Z 215.327,A -85,B 0,C 180,E1 -1582.392,E2 -1582.392} C_VEL
LIN {X 0,Y 587.348,Z 215.326,A -85,B 0,C 180,E1 -1585.653,E2 -1585.653} C_VEL
LIN {X 0,Y 587.345,Z 215.32,A -85,B 0,C 180,E1 -1588.231,E2 -1588.231} C_VEL
LIN {X 0,Y 587.346,Z 215.326,A -85,B 0,C 180,E1 -1590.868,E2 -1590.868} C_VEL
LIN {X 0,Y 587.308,Z 215.326,A -85,B 0,C 180,E1 -1593.83,E2 -1593.83} C_VEL
LIN {X 0,Y 587.312,Z 215.324,A -85,B 0,C 180,E1 -1596.741,E2 -1596.741} C_VEL
LIN {X 0,Y 587.332,Z 215.325,A -85,B 0,C 180,E1 -1599.695,E2 -1599.695} C_VEL
LIN {X 0,Y 587.349,Z 215.324,A -85,B 0,C 180,E1 -1602.594,E2 -1602.594} C_VEL
LIN {X 0,Y 587.345,Z 215.322,A -85,B 0,C 180,E1 -1605.75,E2 -1605.75} C_VEL
LIN {X 0,Y 587.302,Z 215.325,A -85,B 0,C 180,E1 -1608.893,E2 -1608.893} C_VEL
LIN {X 0,Y 587.33,Z 215.324,A -85,B 0,C 180,E1 -1611.744,E2 -1611.744} C_VEL
LIN {X 0,Y 587.322,Z 215.323,A -85,B 0,C 180,E1 -1613.818,E2 -1613.818} C_VEL
LIN {X 0,Y 587.315,Z 215.325,A -85,B 0,C 180,E1 -1615.883,E2 -1615.883} C_VEL
LIN {X 0,Y 587.374,Z 215.321,A -85,B 0,C 180,E1 -1617.943,E2 -1617.943} C_VEL
LIN {X 0,Y 587.378,Z 215.321,A -85,B 0,C 180,E1 -1620,E2 -1620} C_VEL
LIN {X 0,Y 587.346,Z 215.32,A -85,B 0,C 180,E1 -1622.743,E2 -1622.743} C_VEL
LIN {X 0,Y 587.357,Z 215.32,A -85,B 0,C 180,E1 -1625.493,E2 -1625.493} C_VEL
LIN {X 0,Y 587.333,Z 215.327,A -85,B 0,C 180,E1 -1628.256,E2 -1628.256} C_VEL
LIN {X 0,Y 587.355,Z 215.319,A -85,B 0,C 180,E1 -1631.134,E2 -1631.134} C_VEL
LIN {X 0,Y 587.332,Z 215.325,A -85,B 0,C 180,E1 -1633.846,E2 -1633.846} C_VEL
LIN {X 0,Y 587.301,Z 215.33,A -85,B 0,C 180,E1 -1636.796,E2 -1636.796} C_VEL
LIN {X 0,Y 587.294,Z 215.327,A -85,B 0,C 180,E1 -1638.298,E2 -1638.298} C_VEL
LIN {X 0,Y 586.662,Z 215.41,A -85,B 0,C 180,E1 -1638.87,E2 -1638.87} C_VEL
LIN {X 0,Y 583.848,Z 215.757,A -85,B 0,C 180,E1 -1639.799,E2 -1639.799} C_VEL
LIN {X 0,Y 581.439,Z 216.061,A -85,B 0,C 180,E1 -1640.546,E2 -1640.546} C_VEL
LIN {X 0,Y 580.385,Z 216.188,A -85,B 0,C 180,E1 -1641.123,E2 -1641.123} C_VEL
LIN {X 0,Y 580.29,Z 216.199,A -85,B 0,C 180,E1 -1641.318,E2 -1641.318} C_VEL
LIN {X 0,Y 580.303,Z 216.199,A -85,B 0,C 180,E1 -1644.316,E2 -1644.316} C_VEL
LIN {X 0,Y 580.274,Z 216.201,A -85,B 0,C 180,E1 -1646.624,E2 -1646.624} C_VEL
LIN {X 0,Y 580.254,Z 216.203,A -85,B 0,C 180,E1 -1649.775,E2 -1649.775} C_VEL
LIN {X 0,Y 580.301,Z 216.202,A -85,B 0,C 180,E1 -1652.201,E2 -1652.201} C_VEL
LIN {X 0,Y 580.291,Z 216.199,A -85,B 0,C 180,E1 -1654.696,E2 -1654.696} C_VEL
LIN {X 0,Y 580.302,Z 216.202,A -85,B 0,C 180,E1 -1657.268,E2 -1657.268} C_VEL
LIN {X 0,Y 580.293,Z 216.199,A -85,B 0,C 180,E1 -1660.27,E2 -1660.27} C_VEL
LIN {X 0,Y 580.274,Z 216.207,A -85,B 0,C 180,E1 -1662.707,E2 -1662.707} C_VEL
LIN {X 0,Y 580.254,Z 216.205,A -85,B 0,C 180,E1 -1665.611,E2 -1665.611} C_VEL
LIN {X 0,Y 580.262,Z 216.204,A -85,B 0,C 180,E1 -1668.229,E2 -1668.229} C_VEL
LIN {X 0,Y 580.282,Z 216.204,A -85,B 0,C 180,E1 -1670.965,E2 -1670.965} C_VEL
LIN {X 0,Y 580.267,Z 216.202,A -85,B 0,C 180,E1 -1673.596,E2 -1673.596} C_VEL
LIN {X 0,Y 580.176,Z 216.582,A -85,B 0,C 180,E1 -1675.46,E2 -1675.46} C_VEL
LIN {X 0,Y 580.133,Z 219.435,A -85,B 0,C 180,E1 -1677.997,E2 -1677.997} C_VEL
LIN {X 0,Y 580.125,Z 222.432,A -85,B 0,C 180,E1 -1680.722,E2 -1680.722} C_VEL
LIN {X 0,Y 580.079,Z 225.434,A -85,B 0,C 180,E1 -1683.366,E2 -1683.366} C_VEL
LIN {X 0,Y 580.116,Z 228.074,A -85,B 0,C 180,E1 -1685.675,E2 -1685.675} C_VEL
LIN {X 0,Y 580.061,Z 231.689,A -85,B 0,C 180,E1 -1688.686,E2 -1688.686} C_VEL
LIN {X 0,Y 580.032,Z 235.532,A -85,B 0,C 180,E1 -1691.637,E2 -1691.637} C_VEL
LIN {X 0,Y 580.052,Z 239.375,A -85,B 0,C 180,E1 -1694.54,E2 -1694.54} C_VEL
LIN {X 0,Y 580.054,Z 242.258,A -85,B 0,C 180,E1 -1696.691,E2 -1696.691} C_VEL
LIN {X 0,Y 580.061,Z 243.669,A -85,B 0,C 180,E1 -1697.736,E2 -1697.736} C_VEL
LIN {X 0,Y 580.762,Z 249.398,A -85,B 0,C 180,E1 -1697.884,E2 -1697.884} C_VEL
LIN {X 0,Y 580.701,Z 262.446,A -85,B 0,C 180,E1 -1698.26,E2 -1698.26} C_VEL
LIN {X 0,Y 580.624,Z 274.314,A -85,B 0,C 180,E1 -1698.739,E2 -1698.739} C_VEL
LIN {X 0,Y 580.499,Z 286.026,A -85,B 0,C 180,E1 -1699.36,E2 -1699.36} C_VEL
LIN {X 0,Y 580.385,Z 297.663,A -85,B 0,C 180,E1 -1700.151,E2 -1700.151} C_VEL
LIN {X 0,Y 580.308,Z 307.042,A -85,B 0,C 180,E1 -1700.941,E2 -1700.941} C_VEL
LIN {X 0,Y 580.251,Z 315.604,A -85,B 0,C 180,E1 -1701.818,E2 -1701.818} C_VEL
LIN {X 0,Y 580.205,Z 323.918,A -85,B 0,C 180,E1 -1702.868,E2 -1702.868} C_VEL
LIN {X 0,Y 580.14,Z 330.616,A -85,B 0,C 180,E1 -1703.915,E2 -1703.915} C_VEL
LIN {X 0,Y 580.053,Z 336.76,A -85,B 0,C 180,E1 -1705.135,E2 -1705.135} C_VEL
LIN {X 0,Y 580.109,Z 340.749,A -85,B 0,C 180,E1 -1706.179,E2 -1706.179} C_VEL
LIN {X 0,Y 580.043,Z 343.698,A -85,B 0,C 180,E1 -1707.222,E2 -1707.222} C_VEL
LIN {X 0,Y 580.038,Z 345.127,A -85,B 0,C 180,E1 -1707.917,E2 -1707.917} C_VEL
LIN {X 0,Y 580.041,Z 346.755,A -85,B 0,C 180,E1 -1709.306,E2 -1709.306} C_VEL
LIN {X 0,Y 580.038,Z 346.996,A -85,B 0,C 180,E1 -1710,E2 -1710} C_VEL
LIN {X 0,Y 580.04,Z 346.815,A -85,B 0,C 180,E1 -1710.694,E2 -1710.694} C_VEL
LIN {X 0,Y 580.037,Z 345.272,A -85,B 0,C 180,E1 -1712.083,E2 -1712.083} C_VEL
LIN {X 0,Y 580.044,Z 343.911,A -85,B 0,C 180,E1 -1712.778,E2 -1712.778} C_VEL
LIN {X 0,Y 580.109,Z 341.034,A -85,B 0,C 180,E1 -1713.821,E2 -1713.821} C_VEL
LIN {X 0,Y 580.053,Z 337.134,A -85,B 0,C 180,E1 -1714.865,E2 -1714.865} C_VEL
LIN {X 0,Y 580.162,Z 332.102,A -85,B 0,C 180,E1 -1715.91,E2 -1715.91} C_VEL
LIN {X 0,Y 580.158,Z 325.78,A -85,B 0,C 180,E1 -1716.958,E2 -1716.958} C_VEL
LIN {X 0,Y 580.241,Z 317.86,A -85,B 0,C 180,E1 -1718.007,E2 -1718.007} C_VEL
LIN {X 0,Y 580.308,Z 308.011,A -85,B 0,C 180,E1 -1719.058,E2 -1719.058} C_VEL
LIN {X 0,Y 580.404,Z 297.692,A -85,B 0,C 180,E1 -1719.936,E2 -1719.936} C_VEL
LIN {X 0,Y 580.492,Z 286.056,A -85,B 0,C 180,E1 -1720.728,E2 -1720.728} C_VEL
LIN {X 0,Y 580.62,Z 274.408,A -85,B 0,C 180,E1 -1721.347,E2 -1721.347} C_VEL
LIN {X 0,Y 580.672,Z 262.625,A -85,B 0,C 180,E1 -1721.825,E2 -1721.825} C_VEL
LIN {X 0,Y 580.771,Z 249.466,A -85,B 0,C 180,E1 -1722.204,E2 -1722.204} C_VEL
LIN {X 0,Y 580.081,Z 243.671,A -85,B 0,C 180,E1 -1722.352,E2 -1722.352} C_VEL
LIN {X 0,Y 580.044,Z 240.457,A -85,B 0,C 180,E1 -1724.741,E2 -1724.741} C_VEL
LIN {X 0,Y 580.066,Z 237.573,A -85,B 0,C 180,E1 -1726.905,E2 -1726.905} C_VEL
LIN {X 0,Y 580.049,Z 233.728,A -85,B 0,C 180,E1 -1729.831,E2 -1729.831} C_VEL
LIN {X 0,Y 580.038,Z 230.844,A -85,B 0,C 180,E1 -1732.062,E2 -1732.062} C_VEL
LIN {X 0,Y 580.103,Z 227.797,A -85,B 0,C 180,E1 -1734.683,E2 -1734.683} C_VEL
LIN {X 0,Y 580.122,Z 224.692,A -85,B 0,C 180,E1 -1737.41,E2 -1737.41} C_VEL
LIN {X 0,Y 580.143,Z 221.976,A -85,B 0,C 180,E1 -1739.781,E2 -1739.781} C_VEL
LIN {X 0,Y 580.127,Z 219.314,A -85,B 0,C 180,E1 -1742.211,E2 -1742.211} C_VEL
LIN {X 0,Y 580.162,Z 216.504,A -85,B 0,C 180,E1 -1744.705,E2 -1744.705} C_VEL
LIN {X 0,Y 580.264,Z 216.202,A -85,B 0,C 180,E1 -1746.404,E2 -1746.404} C_VEL
LIN {X 0,Y 580.302,Z 216.201,A -85,B 0,C 180,E1 -1749.186,E2 -1749.186} C_VEL
LIN {X 0,Y 580.283,Z 216.2,A -85,B 0,C 180,E1 -1751.769,E2 -1751.769} C_VEL
LIN {X 0,Y 580.249,Z 216.204,A -85,B 0,C 180,E1 -1754.628,E2 -1754.628} C_VEL
LIN {X 0,Y 580.286,Z 216.204,A -85,B 0,C 180,E1 -1757.628,E2 -1757.628} C_VEL
LIN {X 0,Y 580.284,Z 216.2,A -85,B 0,C 180,E1 -1760.066,E2 -1760.066} C_VEL
LIN {X 0,Y 580.301,Z 216.199,A -85,B 0,C 180,E1 -1763.066,E2 -1763.066} C_VEL
LIN {X 0,Y 580.303,Z 216.202,A -85,B 0,C 180,E1 -1766.144,E2 -1766.144} C_VEL
LIN {X 0,Y 580.265,Z 216.201,A -85,B 0,C 180,E1 -1768.614,E2 -1768.614} C_VEL
LIN {X 0,Y 580.282,Z 216.205,A -85,B 0,C 180,E1 -1771.023,E2 -1771.023} C_VEL
LIN {X 0,Y 580.282,Z 216.202,A -85,B 0,C 180,E1 -1774.15,E2 -1774.15} C_VEL
LIN {X 0,Y 580.278,Z 216.205,A -85,B 0,C 180,E1 -1776.442,E2 -1776.442} C_VEL
LIN {X 0,Y 580.276,Z 216.205,A -85,B 0,C 180,E1 -1779.437,E2 -1779.437} C_VEL
LIN {X 0,Y 580.254,Z 216.206,A -85,B 0,C 180,E1 -1781.645,E2 -1781.645} C_VEL
LIN {X 0,Y 580.275,Z 216.204,A -85,B 0,C 180,E1 -1784.547,E2 -1784.547} C_VEL
LIN {X 0,Y 580.299,Z 216.198,A -85,B 0,C 180,E1 -1787.408,E2 -1787.408} C_VEL
LIN {X 0,Y 580.278,Z 216.204,A -85,B 0,C 180,E1 -1790.238,E2 -1790.238} C_VEL
LIN {X 0,Y 580.349,Z 216.198,A -85,B 0,C 180,E1 -1793.227,E2 -1793.227} C_VEL
LIN {X 0,Y 580.239,Z 216.205,A -85,B 0,C 180,E1 -1795.832,E2 -1795.832} C_VEL
LIN {X 0,Y 580.313,Z 216.196,A -85,B 0,C 180,E1 -1797.918,E2 -1797.918} C_VEL
LIN {X 0,Y 580.358,Z 216.191,A -85,B 0,C 180,E1 -1800.694,E2 -1800.694} C_VEL
LIN {X 0,Y 580.279,Z 216.206,A -85,B 0,C 180,E1 -1803.472,E2 -1803.472} C_VEL
LIN {X 0,Y 580.327,Z 216.198,A -85,B 0,C 180,E1 -1805.56,E2 -1805.56} C_VEL
LIN {X 0,Y 580.293,Z 216.199,A -85,B 0,C 180,E1 -1807.656,E2 -1807.656} C_VEL
LIN {X 0,Y 580.278,Z 216.207,A -85,B 0,C 180,E1 -1810.467,E2 -1810.467} C_VEL
LIN {X 0,Y 580.245,Z 216.205,A -85,B 0,C 180,E1 -1813.305,E2 -1813.305} C_VEL
LIN {X 0,Y 580.284,Z 216.205,A -85,B 0,C 180,E1 -1815.453,E2 -1815.453} C_VEL
LIN {X 0,Y 580.295,Z 216.201,A -85,B 0,C 180,E1 -1817.625,E2 -1817.625} C_VEL
LIN {X 0,Y 580.291,Z 216.199,A -85,B 0,C 180,E1 -1819.823,E2 -1819.823} C_VEL
LIN {X 0,Y 580.273,Z 216.204,A -85,B 0,C 180,E1 -1822.053,E2 -1822.053} C_VEL
LIN {X 0,Y 580.26,Z 216.203,A -85,B 0,C 180,E1 -1824.716,E2 -1824.716} C_VEL
LIN {X 0,Y 580.25,Z 216.209,A -85,B 0,C 180,E1 -1827.404,E2 -1827.404} C_VEL
LIN {X 0,Y 580.269,Z 216.202,A -85,B 0,C 180,E1 -1829.774,E2 -1829.774} C_VEL
LIN {X 0,Y 580.303,Z 216.199,A -85,B 0,C 180,E1 -1832.2,E2 -1832.2} C_VEL
LIN {X 0,Y 580.29,Z 216.202,A -85,B 0,C 180,E1 -1834.696,E2 -1834.696} C_VEL
LIN {X 0,Y 580.287,Z 216.201,A -85,B 0,C 180,E1 -1837.269,E2 -1837.269} C_VEL
LIN {X 0,Y 580.274,Z 216.2,A -85,B 0,C 180,E1 -1840.268,E2 -1840.268} C_VEL
LIN {X 0,Y 580.27,Z 216.202,A -85,B 0,C 180,E1 -1843.39,E2 -1843.39} C_VEL
LIN {X 0,Y 580.277,Z 216.204,A -85,B 0,C 180,E1 -1846.61,E2 -1846.61} C_VEL
LIN {X 0,Y 580.299,Z 216.199,A -85,B 0,C 180,E1 -1849.156,E2 -1849.156} C_VEL
LIN {X 0,Y 580.285,Z 216.203,A -85,B 0,C 180,E1 -1851.928,E2 -1851.928} C_VEL
LIN {X 0,Y 580.301,Z 216.33,A -85,B 0,C 180,E1 -1853.504,E2 -1853.504} C_VEL
LIN {X 0,Y 580.734,Z 220.592,A -85,B 0,C 180,E1 -1854.911,E2 -1854.911} C_VEL
LIN {X 0,Y 580.648,Z 228.536,A -85,B 0,C 180,E1 -1857.41,E2 -1857.41} C_VEL
LIN {X 0,Y 580.578,Z 237.803,A -85,B 0,C 180,E1 -1860.244,E2 -1860.244} C_VEL
LIN {X 0,Y 580.473,Z 247.07,A -85,B 0,C 180,E1 -1862.998,E2 -1862.998} C_VEL
LIN {X 0,Y 580.393,Z 256.338,A -85,B 0,C 180,E1 -1865.688,E2 -1865.688} C_VEL
LIN {X 0,Y 580.36,Z 265.605,A -85,B 0,C 180,E1 -1868.325,E2 -1868.325} C_VEL
LIN {X 0,Y 580.259,Z 276.196,A -85,B 0,C 180,E1 -1871.279,E2 -1871.279} C_VEL
LIN {X 0,Y 580.211,Z 285.464,A -85,B 0,C 180,E1 -1873.824,E2 -1873.824} C_VEL
LIN {X 0,Y 580.175,Z 296.055,A -85,B 0,C 180,E1 -1876.694,E2 -1876.694} C_VEL
LIN {X 0,Y 580.119,Z 299.53,A -85,B 0,C 180,E1 -1877.627,E2 -1877.627} C_VEL
LIN {X 0,Y 580.799,Z 305.231,A -85,B 0,C 180,E1 -1877.752,E2 -1877.752} C_VEL
LIN {X 0,Y 580.716,Z 318.497,A -85,B 0,C 180,E1 -1878.083,E2 -1878.083} C_VEL
LIN {X 0,Y 580.598,Z 330.639,A -85,B 0,C 180,E1 -1878.528,E2 -1878.528} C_VEL
LIN {X 0,Y 580.507,Z 342.21,A -85,B 0,C 180,E1 -1879.096,E2 -1879.096} C_VEL
LIN {X 0,Y 580.446,Z 353.477,A -85,B 0,C 180,E1 -1879.8,E2 -1879.8} C_VEL
LIN {X 0,Y 580.352,Z 363.647,A -85,B 0,C 180,E1 -1880.591,E2 -1880.591} C_VEL
LIN {X 0,Y 580.279,Z 372.788,A -85,B 0,C 180,E1 -1881.468,E2 -1881.468} C_VEL
LIN {X 0,Y 580.199,Z 381.691,A -85,B 0,C 180,E1 -1882.518,E2 -1882.518} C_VEL
LIN {X 0,Y 580.12,Z 388.466,A -85,B 0,C 180,E1 -1883.505,E2 -1883.505} C_VEL
LIN {X 0,Y 580.139,Z 393.681,A -85,B 0,C 180,E1 -1884.439,E2 -1884.439} C_VEL
LIN {X 0,Y 580.108,Z 398.372,A -85,B 0,C 180,E1 -1885.483,E2 -1885.483} C_VEL
LIN {X 0,Y 580.123,Z 401.957,A -85,B 0,C 180,E1 -1886.527,E2 -1886.527} C_VEL
LIN {X 0,Y 580.043,Z 403.809,A -85,B 0,C 180,E1 -1887.222,E2 -1887.222} C_VEL
LIN {X 0,Y 580.04,Z 405.201,A -85,B 0,C 180,E1 -1887.917,E2 -1887.917} C_VEL
LIN {X 0,Y 580.04,Z 406.784,A -85,B 0,C 180,E1 -1889.306,E2 -1889.306} C_VEL
LIN {X 0,Y 580.037,Z 407,A -85,B 0,C 180,E1 -1890,E2 -1890} C_VEL
LIN {X 0,Y 580.047,Z 406.185,A -85,B 0,C 180,E1 -1891.389,E2 -1891.389} C_VEL
LIN {X 0,Y 580.04,Z 405.201,A -85,B 0,C 180,E1 -1892.083,E2 -1892.083} C_VEL
LIN {X 0,Y 580.043,Z 403.809,A -85,B 0,C 180,E1 -1892.778,E2 -1892.778} C_VEL
LIN {X 0,Y 580.11,Z 400.896,A -85,B 0,C 180,E1 -1893.821,E2 -1893.821} C_VEL
LIN {X 0,Y 580.053,Z 396.949,A -85,B 0,C 180,E1 -1894.865,E2 -1894.865} C_VEL
LIN {X 0,Y 580.139,Z 390.877,A -85,B 0,C 180,E1 -1896.085,E2 -1896.085} C_VEL
LIN {X 0,Y 580.184,Z 384.235,A -85,B 0,C 180,E1 -1897.133,E2 -1897.133} C_VEL
LIN {X 0,Y 580.25,Z 375.988,A -85,B 0,C 180,E1 -1898.182,E2 -1898.182} C_VEL
LIN {X 0,Y 580.308,Z 367.535,A -85,B 0,C 180,E1 -1899.059,E2 -1899.059} C_VEL
LIN {X 0,Y 580.412,Z 357.091,A -85,B 0,C 180,E1 -1899.936,E2 -1899.936} C_VEL
LIN {X 0,Y 580.454,Z 346.756,A -85,B 0,C 180,E1 -1900.641,E2 -1900.641} C_VEL
LIN {X 0,Y 580.564,Z 335.59,A -85,B 0,C 180,E1 -1901.248,E2 -1901.248} C_VEL
LIN {X 0,Y 580.637,Z 323.762,A -85,B 0,C 180,E1 -1901.742,E2 -1901.742} C_VEL
LIN {X 0,Y 580.779,Z 310.343,A -85,B 0,C 180,E1 -1902.137,E2 -1902.137} C_VEL
LIN {X 0,Y 580.589,Z 302.483,A -85,B 0,C 180,E1 -1902.305,E2 -1902.305} C_VEL
LIN {X 0,Y 580.119,Z 299.53,A -85,B 0,C 180,E1 -1902.373,E2 -1902.373} C_VEL
LIN {X 0,Y 580.216,Z 289.435,A -85,B 0,C 180,E1 -1905.095,E2 -1905.095} C_VEL
LIN {X 0,Y 580.248,Z 278.843,A -85,B 0,C 180,E1 -1907.991,E2 -1907.991} C_VEL
LIN {X 0,Y 580.345,Z 268.49,A -85,B 0,C 180,E1 -1910.865,E2 -1910.865} C_VEL
LIN {X 0,Y 580.408,Z 258.985,A -85,B 0,C 180,E1 -1913.553,E2 -1913.553} C_VEL
LIN {X 0,Y 580.485,Z 249.218,A -85,B 0,C 180,E1 -1916.372,E2 -1916.372} C_VEL
LIN {X 0,Y 580.516,Z 240.45,A -85,B 0,C 180,E1 -1918.964,E2 -1918.964} C_VEL
LIN {X 0,Y 580.657,Z 231.33,A -85,B 0,C 180,E1 -1921.725,E2 -1921.725} C_VEL
LIN {X 0,Y 580.713,Z 223.319,A -85,B 0,C 180,E1 -1924.222,E2 -1924.222} C_VEL
LIN {X 0,Y 580.635,Z 218.373,A -85,B 0,C 180,E1 -1925.809,E2 -1925.809} C_VEL
LIN {X 0,Y 580.281,Z 216.207,A -85,B 0,C 180,E1 -1926.592,E2 -1926.592} C_VEL
LIN {X 0,Y 580.291,Z 216.2,A -85,B 0,C 180,E1 -1929.184,E2 -1929.184} C_VEL
LIN {X 0,Y 580.284,Z 216.205,A -85,B 0,C 180,E1 -1931.769,E2 -1931.769} C_VEL
LIN {X 0,Y 580.252,Z 216.204,A -85,B 0,C 180,E1 -1934.628,E2 -1934.628} C_VEL
LIN {X 0,Y 580.264,Z 216.207,A -85,B 0,C 180,E1 -1937.292,E2 -1937.292} C_VEL
LIN {X 0,Y 580.269,Z 216.202,A -85,B 0,C 180,E1 -1940.065,E2 -1940.065} C_VEL
LIN {X 0,Y 580.279,Z 216.2,A -85,B 0,C 180,E1 -1943.069,E2 -1943.069} C_VEL
LIN {X 0,Y 580.318,Z 216.197,A -85,B 0,C 180,E1 -1946.145,E2 -1946.145} C_VEL
LIN {X 0,Y 580.277,Z 216.202,A -85,B 0,C 180,E1 -1948.614,E2 -1948.614} C_VEL
LIN {X 0,Y 580.284,Z 216.204,A -85,B 0,C 180,E1 -1951.023,E2 -1951.023} C_VEL
LIN {X 0,Y 580.255,Z 216.209,A -85,B 0,C 180,E1 -1954.149,E2 -1954.149} C_VEL
LIN {X 0,Y 580.292,Z 216.2,A -85,B 0,C 180,E1 -1957.197,E2 -1957.197} C_VEL
LIN {X 0,Y 580.279,Z 216.207,A -85,B 0,C 180,E1 -1959.437,E2 -1959.437} C_VEL
LIN {X 0,Y 580.271,Z 216.202,A -85,B 0,C 180,E1 -1961.645,E2 -1961.645} C_VEL
LIN {X 0,Y 580.269,Z 216.202,A -85,B 0,C 180,E1 -1963.825,E2 -1963.825} C_VEL
LIN {X 0,Y 580.315,Z 216.2,A -85,B 0,C 180,E1 -1965.983,E2 -1965.983} C_VEL
LIN {X 0,Y 580.272,Z 216.2,A -85,B 0,C 180,E1 -1968.826,E2 -1968.826} C_VEL
LIN {X 0,Y 580.302,Z 216.2,A -85,B 0,C 180,E1 -1971.644,E2 -1971.644} C_VEL
LIN {X 0,Y 580.281,Z 216.2,A -85,B 0,C 180,E1 -1973.742,E2 -1973.742} C_VEL
LIN {X 0,Y 580.271,Z 216.202,A -85,B 0,C 180,E1 -1975.833,E2 -1975.833} C_VEL
LIN {X 0,Y 580.344,Z 216.196,A -85,B 0,C 180,E1 -1977.918,E2 -1977.918} C_VEL
LIN {X 0,Y 580.348,Z 216.197,A -85,B 0,C 180,E1 -1980,E2 -1980} C_VEL
LIN {X 0,Y 580.316,Z 216.196,A -85,B 0,C 180,E1 -1982.777,E2 -1982.777} C_VEL
LIN {X 0,Y 580.322,Z 216.196,A -85,B 0,C 180,E1 -1985.56,E2 -1985.56} C_VEL
LIN {X 0,Y 580.324,Z 216.195,A -85,B 0,C 180,E1 -1987.655,E2 -1987.655} C_VEL
LIN {X 0,Y 580.3,Z 216.201,A -85,B 0,C 180,E1 -1990.467,E2 -1990.467} C_VEL
LIN {X 0,Y 580.3,Z 216.198,A -85,B 0,C 180,E1 -1992.592,E2 -1992.592} C_VEL
LIN {X 0,Y 580.275,Z 216.205,A -85,B 0,C 180,E1 -1995.453,E2 -1995.453} C_VEL
LIN {X 0,Y 580.252,Z 216.206,A -85,B 0,C 180,E1 -1998.356,E2 -1998.356} C_VEL
LIN {X 0,Y 580.307,Z 216.197,A -85,B 0,C 180,E1 -2001.165,E2 -2001.165} C_VEL
LIN {X 0,Y 580.29,Z 216.199,A -85,B 0,C 180,E1 -2001.318,E2 -2001.318} C_VEL
LIN {X 0,Y 579.59,Z 216.291,A -85,B 0,C 180,E1 -2001.897,E2 -2001.897} C_VEL
LIN {X 0,Y 576.711,Z 216.648,A -85,B 0,C 180,E1 -2002.837,E2 -2002.837} C_VEL
LIN {X 0,Y 574.316,Z 216.948,A -85,B 0,C 180,E1 -2003.593,E2 -2003.593} C_VEL
LIN {X 0,Y 573.318,Z 217.07,A -85,B 0,C 180,E1 -2004.177,E2 -2004.177} C_VEL
LIN {X 0,Y 573.253,Z 217.076,A -85,B 0,C 180,E1 -2004.375,E2 -2004.375} C_VEL
LIN {X 0,Y 573.209,Z 217.085,A -85,B 0,C 180,E1 -2006.978,E2 -2006.978} C_VEL
LIN {X 0,Y 573.216,Z 217.081,A -85,B 0,C 180,E1 -2009.482,E2 -2009.482} C_VEL
LIN {X 0,Y 573.257,Z 217.078,A -85,B 0,C 180,E1 -2012.645,E2 -2012.645} C_VEL
LIN {X 0,Y 573.21,Z 217.082,A -85,B 0,C 180,E1 -2015.188,E2 -2015.188} C_VEL
LIN {X 0,Y 573.238,Z 217.081,A -85,B 0,C 180,E1 -2017.808,E2 -2017.808} C_VEL
LIN {X 0,Y 573.249,Z 217.079,A -85,B 0,C 180,E1 -2020.525,E2 -2020.525} C_VEL
LIN {X 0,Y 573.21,Z 217.081,A -85,B 0,C 180,E1 -2023.362,E2 -2023.362} C_VEL
LIN {X 0,Y 573.21,Z 217.084,A -85,B 0,C 180,E1 -2026.335,E2 -2026.335} C_VEL
LIN {X 0,Y 573.223,Z 217.079,A -85,B 0,C 180,E1 -2028.542,E2 -2028.542} C_VEL
LIN {X 0,Y 573.246,Z 217.082,A -85,B 0,C 180,E1 -2031.298,E2 -2031.298} C_VEL
LIN {X 0,Y 573.192,Z 217.084,A -85,B 0,C 180,E1 -2034.022,E2 -2034.022} C_VEL
LIN {X 0,Y 573.103,Z 217.101,A -85,B 0,C 180,E1 -2035.248,E2 -2035.248} C_VEL
LIN {X 0,Y 573.065,Z 219.924,A -85,B 0,C 180,E1 -2037.802,E2 -2037.802} C_VEL
LIN {X 0,Y 573.074,Z 222.888,A -85,B 0,C 180,E1 -2040.543,E2 -2040.543} C_VEL
LIN {X 0,Y 573.025,Z 225.651,A -85,B 0,C 180,E1 -2043.012,E2 -2043.012} C_VEL
LIN {X 0,Y 573.029,Z 228.324,A -85,B 0,C 180,E1 -2045.355,E2 -2045.355} C_VEL
LIN {X 0,Y 572.967,Z 231.806,A -85,B 0,C 180,E1 -2048.409,E2 -2048.409} C_VEL
LIN {X 0,Y 572.971,Z 234.776,A -85,B 0,C 180,E1 -2050.818,E2 -2050.818} C_VEL
LIN {X 0,Y 572.966,Z 238.415,A -85,B 0,C 180,E1 -2053.613,E2 -2053.613} C_VEL
LIN {X 0,Y 572.981,Z 242.259,A -85,B 0,C 180,E1 -2056.523,E2 -2056.523} C_VEL
LIN {X 0,Y 572.999,Z 243.67,A -85,B 0,C 180,E1 -2057.583,E2 -2057.583} C_VEL
LIN {X 0,Y 573.819,Z 250.335,A -85,B 0,C 180,E1 -2057.758,E2 -2057.758} C_VEL
LIN {X 0,Y 573.717,Z 263.758,A -85,B 0,C 180,E1 -2058.16,E2 -2058.16} C_VEL
LIN {X 0,Y 573.629,Z 276.284,A -85,B 0,C 180,E1 -2058.695,E2 -2058.695} C_VEL
LIN {X 0,Y 573.507,Z 287.462,A -85,B 0,C 180,E1 -2059.319,E2 -2059.319} C_VEL
LIN {X 0,Y 573.345,Z 298.832,A -85,B 0,C 180,E1 -2060.118,E2 -2060.118} C_VEL
LIN {X 0,Y 573.28,Z 308.883,A -85,B 0,C 180,E1 -2061.007,E2 -2061.007} C_VEL
LIN {X 0,Y 573.161,Z 318.585,A -85,B 0,C 180,E1 -2062.071,E2 -2062.071} C_VEL
LIN {X 0,Y 573.093,Z 326.523,A -85,B 0,C 180,E1 -2063.162,E2 -2063.162} C_VEL
LIN {X 0,Y 573.07,Z 333.448,A -85,B 0,C 180,E1 -2064.37,E2 -2064.37} C_VEL
LIN {X 0,Y 573.028,Z 338.19,A -85,B 0,C 180,E1 -2065.427,E2 -2065.427} C_VEL
LIN {X 0,Y 573.022,Z 341.823,A -85,B 0,C 180,E1 -2066.484,E2 -2066.484} C_VEL
LIN {X 0,Y 572.959,Z 343.7,A -85,B 0,C 180,E1 -2067.188,E2 -2067.188} C_VEL
LIN {X 0,Y 572.938,Z 345.127,A -85,B 0,C 180,E1 -2067.891,E2 -2067.891} C_VEL
LIN {X 0,Y 572.941,Z 346.755,A -85,B 0,C 180,E1 -2069.297,E2 -2069.297} C_VEL
LIN {X 0,Y 572.938,Z 346.996,A -85,B 0,C 180,E1 -2070,E2 -2070} C_VEL
LIN {X 0,Y 572.94,Z 346.815,A -85,B 0,C 180,E1 -2070.703,E2 -2070.703} C_VEL
LIN {X 0,Y 572.937,Z 345.27,A -85,B 0,C 180,E1 -2072.109,E2 -2072.109} C_VEL
LIN {X 0,Y 572.96,Z 343.909,A -85,B 0,C 180,E1 -2072.812,E2 -2072.812} C_VEL
LIN {X 0,Y 573.014,Z 341.032,A -85,B 0,C 180,E1 -2073.868,E2 -2073.868} C_VEL
LIN {X 0,Y 572.963,Z 337.132,A -85,B 0,C 180,E1 -2074.926,E2 -2074.926} C_VEL
LIN {X 0,Y 573.075,Z 332.1,A -85,B 0,C 180,E1 -2075.983,E2 -2075.983} C_VEL
LIN {X 0,Y 573.083,Z 325.776,A -85,B 0,C 180,E1 -2077.044,E2 -2077.044} C_VEL
LIN {X 0,Y 573.175,Z 317.855,A -85,B 0,C 180,E1 -2078.106,E2 -2078.106} C_VEL
LIN {X 0,Y 573.287,Z 308.005,A -85,B 0,C 180,E1 -2079.17,E2 -2079.17} C_VEL
LIN {X 0,Y 573.405,Z 297.686,A -85,B 0,C 180,E1 -2080.059,E2 -2080.059} C_VEL
LIN {X 0,Y 573.489,Z 286.136,A -85,B 0,C 180,E1 -2080.855,E2 -2080.855} C_VEL
LIN {X 0,Y 573.658,Z 275.2,A -85,B 0,C 180,E1 -2081.449,E2 -2081.449} C_VEL
LIN {X 0,Y 573.722,Z 262.61,A -85,B 0,C 180,E1 -2081.97,E2 -2081.97} C_VEL
LIN {X 0,Y 573.823,Z 248.984,A -85,B 0,C 180,E1 -2082.365,E2 -2082.365} C_VEL
LIN {X 0,Y 572.962,Z 243.67,A -85,B 0,C 180,E1 -2082.508,E2 -2082.508} C_VEL
LIN {X 0,Y 572.957,Z 240.456,A -85,B 0,C 180,E1 -2084.927,E2 -2084.927} C_VEL
LIN {X 0,Y 572.975,Z 237.572,A -85,B 0,C 180,E1 -2087.12,E2 -2087.12} C_VEL
LIN {X 0,Y 572.977,Z 233.727,A -85,B 0,C 180,E1 -2090.087,E2 -2090.087} C_VEL
LIN {X 0,Y 572.991,Z 230.198,A -85,B 0,C 180,E1 -2093.11,E2 -2093.11} C_VEL
LIN {X 0,Y 573.017,Z 227.542,A -85,B 0,C 180,E1 -2095.421,E2 -2095.421} C_VEL
LIN {X 0,Y 573.076,Z 224.633,A -85,B 0,C 180,E1 -2097.995,E2 -2097.995} C_VEL
LIN {X 0,Y 573.102,Z 221.46,A -85,B 0,C 180,E1 -2100.86,E2 -2100.86} C_VEL
LIN {X 0,Y 573.124,Z 218.554,A -85,B 0,C 180,E1 -2103.503,E2 -2103.503} C_VEL
LIN {X 0,Y 573.099,Z 217.142,A -85,B 0,C 180,E1 -2104.751,E2 -2104.751} C_VEL
LIN {X 0,Y 573.255,Z 217.082,A -85,B 0,C 180,E1 -2107.166,E2 -2107.166} C_VEL
LIN {X 0,Y 573.244,Z 217.077,A -85,B 0,C 180,E1 -2109.608,E2 -2109.608} C_VEL
LIN {X 0,Y 573.238,Z 217.08,A -85,B 0,C 180,E1 -2112.641,E2 -2112.641} C_VEL
LIN {X 0,Y 573.219,Z 217.085,A -85,B 0,C 180,E1 -2115.665,E2 -2115.665} C_VEL
LIN {X 0,Y 573.221,Z 217.08,A -85,B 0,C 180,E1 -2118.542,E2 -2118.542} C_VEL
LIN {X 0,Y 573.242,Z 217.079,A -85,B 0,C 180,E1 -2121.298,E2 -2121.298} C_VEL
LIN {X 0,Y 573.217,Z 217.084,A -85,B 0,C 180,E1 -2124.018,E2 -2124.018} C_VEL
LIN {X 0,Y 573.241,Z 217.078,A -85,B 0,C 180,E1 -2126.516,E2 -2126.516} C_VEL
LIN {X 0,Y 573.215,Z 217.083,A -85,B 0,C 180,E1 -2129.121,E2 -2129.121} C_VEL
LIN {X 0,Y 573.204,Z 217.085,A -85,B 0,C 180,E1 -2131.434,E2 -2131.434} C_VEL
LIN {X 0,Y 573.252,Z 217.082,A -85,B 0,C 180,E1 -2134.59,E2 -2134.59} C_VEL
LIN {X 0,Y 573.24,Z 217.081,A -85,B 0,C 180,E1 -2137.662,E2 -2137.662} C_VEL
LIN {X 0,Y 573.27,Z 217.073,A -85,B 0,C 180,E1 -2140.67,E2 -2140.67} C_VEL
LIN {X 0,Y 573.222,Z 217.08,A -85,B 0,C 180,E1 -2143.621,E2 -2143.621} C_VEL
LIN {X 0,Y 573.213,Z 217.087,A -85,B 0,C 180,E1 -2146.529,E2 -2146.529} C_VEL
LIN {X 0,Y 573.267,Z 217.075,A -85,B 0,C 180,E1 -2148.745,E2 -2148.745} C_VEL
LIN {X 0,Y 573.259,Z 217.081,A -85,B 0,C 180,E1 -2151.54,E2 -2151.54} C_VEL
LIN {X 0,Y 573.233,Z 217.081,A -85,B 0,C 180,E1 -2153.665,E2 -2153.665} C_VEL
LIN {X 0,Y 573.197,Z 217.082,A -85,B 0,C 180,E1 -2155.781,E2 -2155.781} C_VEL
LIN {X 0,Y 573.287,Z 217.071,A -85,B 0,C 180,E1 -2157.892,E2 -2157.892} C_VEL
LIN {X 0,Y 573.329,Z 217.067,A -85,B 0,C 180,E1 -2160.702,E2 -2160.702} C_VEL
LIN {X 0,Y 573.306,Z 217.069,A -85,B 0,C 180,E1 -2162.811,E2 -2162.811} C_VEL
LIN {X 0,Y 573.293,Z 217.074,A -85,B 0,C 180,E1 -2165.628,E2 -2165.628} C_VEL
LIN {X 0,Y 573.247,Z 217.08,A -85,B 0,C 180,E1 -2168.46,E2 -2168.46} C_VEL
LIN {X 0,Y 573.238,Z 217.077,A -85,B 0,C 180,E1 -2171.313,E2 -2171.313} C_VEL
LIN {X 0,Y 573.27,Z 217.074,A -85,B 0,C 180,E1 -2174.418,E2 -2174.418} C_VEL
LIN {X 0,Y 573.262,Z 217.08,A -85,B 0,C 180,E1 -2177.112,E2 -2177.112} C_VEL
LIN {X 0,Y 573.246,Z 217.077,A -85,B 0,C 180,E1 -2180.077,E2 -2180.077} C_VEL
LIN {X 0,Y 573.236,Z 217.085,A -85,B 0,C 180,E1 -2182.338,E2 -2182.338} C_VEL
LIN {X 0,Y 573.212,Z 217.082,A -85,B 0,C 180,E1 -2185.412,E2 -2185.412} C_VEL
LIN {X 0,Y 573.203,Z 217.083,A -85,B 0,C 180,E1 -2188.019,E2 -2188.019} C_VEL
LIN {X 0,Y 573.235,Z 217.078,A -85,B 0,C 180,E1 -2190.177,E2 -2190.177} C_VEL
LIN {X 0,Y 573.258,Z 217.081,A -85,B 0,C 180,E1 -2192.645,E2 -2192.645} C_VEL
LIN {X 0,Y 573.208,Z 217.081,A -85,B 0,C 180,E1 -2195.188,E2 -2195.188} C_VEL
LIN {X 0,Y 573.229,Z 217.085,A -85,B 0,C 180,E1 -2197.808,E2 -2197.808} C_VEL
LIN {X 0,Y 573.23,Z 217.078,A -85,B 0,C 180,E1 -2200.527,E2 -2200.527} C_VEL
LIN {X 0,Y 573.238,Z 217.077,A -85,B 0,C 180,E1 -2203.668,E2 -2203.668} C_VEL
LIN {X 0,Y 573.239,Z 217.081,A -85,B 0,C 180,E1 -2206.641,E2 -2206.641} C_VEL
LIN {X 0,Y 573.247,Z 217.081,A -85,B 0,C 180,E1 -2209.475,E2 -2209.475} C_VEL
LIN {X 0,Y 573.228,Z 217.081,A -85,B 0,C 180,E1 -2212.192,E2 -2212.192} C_VEL
LIN {X 0,Y 573.288,Z 217.283,A -85,B 0,C 180,E1 -2213.3,E2 -2213.3} C_VEL
LIN {X 0,Y 573.789,Z 221.916,A -85,B 0,C 180,E1 -2214.853,E2 -2214.853} C_VEL
LIN {X 0,Y 573.703,Z 230.87,A -85,B 0,C 180,E1 -2217.701,E2 -2217.701} C_VEL
LIN {X 0,Y 573.566,Z 240.451,A -85,B 0,C 180,E1 -2220.651,E2 -2220.651} C_VEL
LIN {X 0,Y 573.483,Z 249.819,A -85,B 0,C 180,E1 -2223.459,E2 -2223.459} C_VEL
LIN {X 0,Y 573.397,Z 258.986,A -85,B 0,C 180,E1 -2226.142,E2 -2226.142} C_VEL
LIN {X 0,Y 573.278,Z 267.919,A -85,B 0,C 180,E1 -2228.703,E2 -2228.703} C_VEL
LIN {X 0,Y 573.202,Z 277.52,A -85,B 0,C 180,E1 -2231.411,E2 -2231.411} C_VEL
LIN {X 0,Y 573.158,Z 286.788,A -85,B 0,C 180,E1 -2233.985,E2 -2233.985} C_VEL
LIN {X 0,Y 573.091,Z 297.379,A -85,B 0,C 180,E1 -2236.887,E2 -2236.887} C_VEL
LIN {X 0,Y 573.078,Z 299.53,A -85,B 0,C 180,E1 -2237.472,E2 -2237.472} C_VEL
LIN {X 0,Y 573.862,Z 306.372,A -85,B 0,C 180,E1 -2237.624,E2 -2237.624} C_VEL
LIN {X 0,Y 573.774,Z 318.497,A -85,B 0,C 180,E1 -2237.937,E2 -2237.937} C_VEL
LIN {X 0,Y 573.642,Z 330.527,A -85,B 0,C 180,E1 -2238.382,E2 -2238.382} C_VEL
LIN {X 0,Y 573.524,Z 342.62,A -85,B 0,C 180,E1 -2238.985,E2 -2238.985} C_VEL
LIN {X 0,Y 573.442,Z 353.478,A -85,B 0,C 180,E1 -2239.674,E2 -2239.674} C_VEL
LIN {X 0,Y 573.307,Z 363.647,A -85,B 0,C 180,E1 -2240.474,E2 -2240.474} C_VEL
LIN {X 0,Y 573.215,Z 372.788,A -85,B 0,C 180,E1 -2241.362,E2 -2241.362} C_VEL
LIN {X 0,Y 573.142,Z 381.691,A -85,B 0,C 180,E1 -2242.425,E2 -2242.425} C_VEL
LIN {X 0,Y 573.051,Z 388.405,A -85,B 0,C 180,E1 -2243.415,E2 -2243.415} C_VEL
LIN {X 0,Y 573.07,Z 393.681,A -85,B 0,C 180,E1 -2244.37,E2 -2244.37} C_VEL
LIN {X 0,Y 573.028,Z 398.372,A -85,B 0,C 180,E1 -2245.428,E2 -2245.428} C_VEL
LIN {X 0,Y 573.022,Z 401.957,A -85,B 0,C 180,E1 -2246.484,E2 -2246.484} C_VEL
LIN {X 0,Y 572.959,Z 403.809,A -85,B 0,C 180,E1 -2247.188,E2 -2247.188} C_VEL
LIN {X 0,Y 572.94,Z 405.201,A -85,B 0,C 180,E1 -2247.891,E2 -2247.891} C_VEL
LIN {X 0,Y 572.94,Z 406.784,A -85,B 0,C 180,E1 -2249.297,E2 -2249.297} C_VEL
LIN {X 0,Y 572.938,Z 407,A -85,B 0,C 180,E1 -2250,E2 -2250} C_VEL
LIN {X 0,Y 572.946,Z 406.185,A -85,B 0,C 180,E1 -2251.406,E2 -2251.406} C_VEL
LIN {X 0,Y 572.94,Z 405.201,A -85,B 0,C 180,E1 -2252.109,E2 -2252.109} C_VEL
LIN {X 0,Y 572.959,Z 403.809,A -85,B 0,C 180,E1 -2252.812,E2 -2252.812} C_VEL
LIN {X 0,Y 573.015,Z 400.896,A -85,B 0,C 180,E1 -2253.868,E2 -2253.868} C_VEL
LIN {X 0,Y 572.963,Z 396.949,A -85,B 0,C 180,E1 -2254.926,E2 -2254.926} C_VEL
LIN {X 0,Y 573.065,Z 390.877,A -85,B 0,C 180,E1 -2256.16,E2 -2256.16} C_VEL
LIN {X 0,Y 573.119,Z 384.235,A -85,B 0,C 180,E1 -2257.221,E2 -2257.221} C_VEL
LIN {X 0,Y 573.201,Z 375.988,A -85,B 0,C 180,E1 -2258.283,E2 -2258.283} C_VEL
LIN {X 0,Y 573.287,Z 367.535,A -85,B 0,C 180,E1 -2259.17,E2 -2259.17} C_VEL
LIN {X 0,Y 573.405,Z 357.092,A -85,B 0,C 180,E1 -2260.059,E2 -2260.059} C_VEL
LIN {X 0,Y 573.519,Z 345.536,A -85,B 0,C 180,E1 -2260.847,E2 -2260.847} C_VEL
LIN {X 0,Y 573.609,Z 333.875,A -85,B 0,C 180,E1 -2261.466,E2 -2261.466} C_VEL
LIN {X 0,Y 573.766,Z 321.17,A -85,B 0,C 180,E1 -2261.974,E2 -2261.974} C_VEL
LIN {X 0,Y 573.863,Z 308.514,A -85,B 0,C 180,E1 -2262.331,E2 -2262.331} C_VEL
LIN {X 0,Y 573.569,Z 302.639,A -85,B 0,C 180,E1 -2262.455,E2 -2262.455} C_VEL
LIN {X 0,Y 573.078,Z 299.53,A -85,B 0,C 180,E1 -2262.528,E2 -2262.528} C_VEL
LIN {X 0,Y 573.156,Z 289.435,A -85,B 0,C 180,E1 -2265.286,E2 -2265.286} C_VEL
LIN {X 0,Y 573.207,Z 278.843,A -85,B 0,C 180,E1 -2268.219,E2 -2268.219} C_VEL
LIN {X 0,Y 573.31,Z 269.576,A -85,B 0,C 180,E1 -2270.824,E2 -2270.824} C_VEL
LIN {X 0,Y 573.374,Z 260.31,A -85,B 0,C 180,E1 -2273.476,E2 -2273.476} C_VEL
LIN {X 0,Y 573.455,Z 251.041,A -85,B 0,C 180,E1 -2276.181,E2 -2276.181} C_VEL
LIN {X 0,Y 573.519,Z 241.774,A -85,B 0,C 180,E1 -2278.95,E2 -2278.95} C_VEL
LIN {X 0,Y 573.695,Z 232.507,A -85,B 0,C 180,E1 -2281.788,E2 -2281.788} C_VEL
LIN {X 0,Y 573.777,Z 224.563,A -85,B 0,C 180,E1 -2284.294,E2 -2284.294} C_VEL
LIN {X 0,Y 573.602,Z 219.234,A -85,B 0,C 180,E1 -2286.035,E2 -2286.035} C_VEL
LIN {X 0,Y 573.239,Z 217.085,A -85,B 0,C 180,E1 -2286.814,E2 -2286.814} C_VEL
LIN {X 0,Y 573.238,Z 217.079,A -85,B 0,C 180,E1 -2289.608,E2 -2289.608} C_VEL
LIN {X 0,Y 573.244,Z 217.078,A -85,B 0,C 180,E1 -2292.642,E2 -2292.642} C_VEL
LIN {X 0,Y 573.226,Z 217.083,A -85,B 0,C 180,E1 -2295.665,E2 -2295.665} C_VEL
